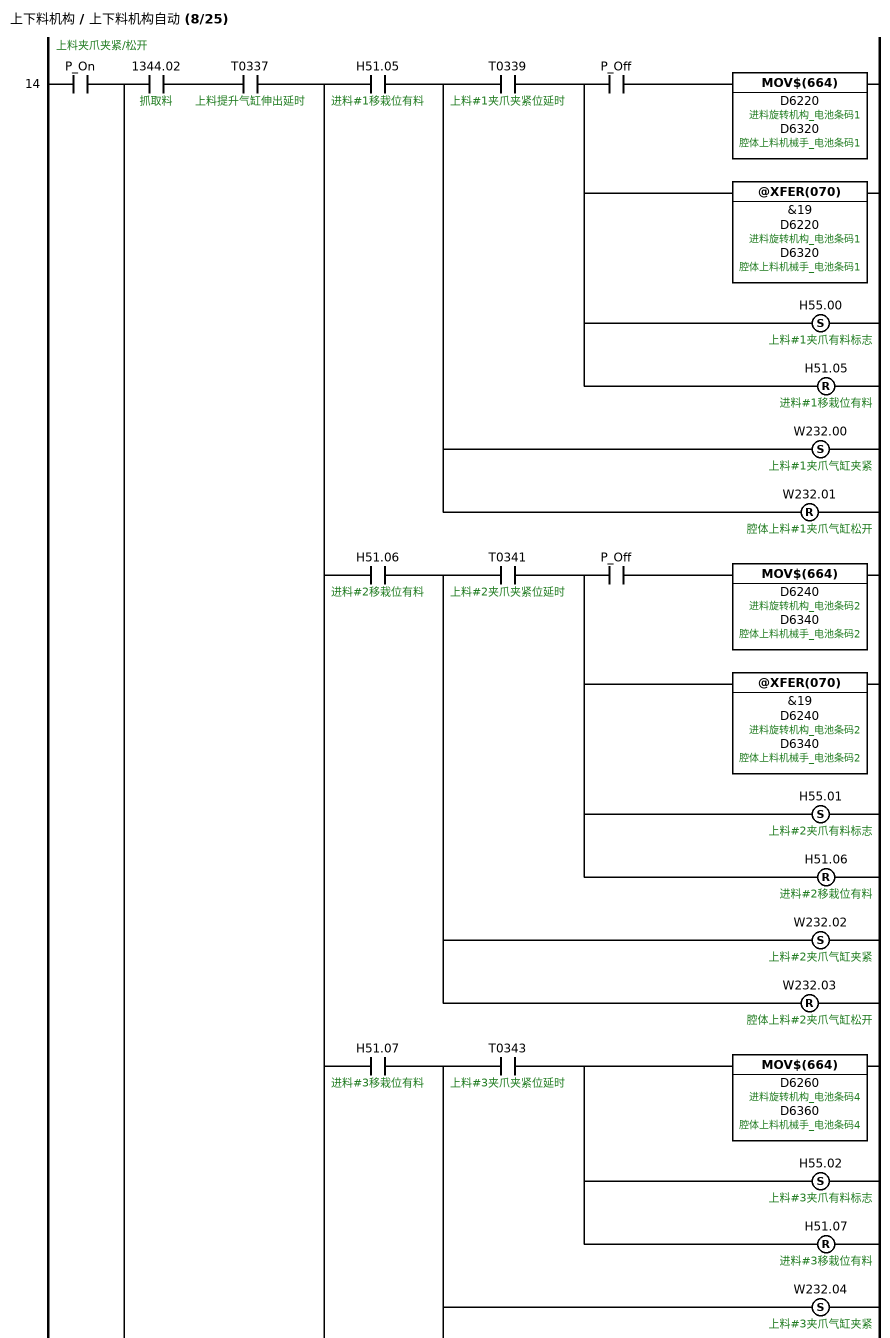
; [picture p168: 上下料机构 / 上下料机构自动, rungs 14-14]

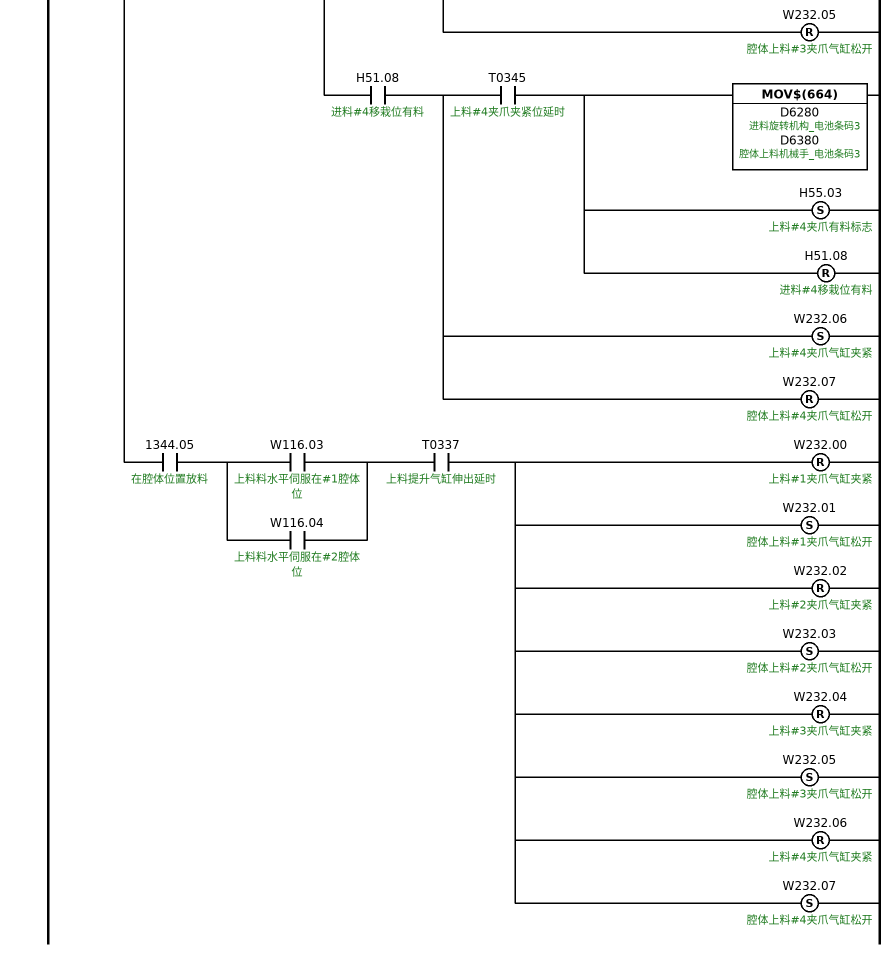
; rung 14: 上料夹爪夹紧/松开
LD P_On
OUT TR0
AND 1344.02  ; 抓取料
AND T0337  ; 上料提升气缸伸出延时
OUT TR1
AND H51.05  ; 进料#1移栽位有料
OUT TR2
AND T0339  ; 上料#1夹爪夹紧位延时
OUT TR3
AND P_Off
MOV$(664) D6220 D6320  ; 进料旋转机构_电池条码1, 腔体上料机械手_电池条码1
LD TR3
@XFER(070) &19 D6220 D6320  ; 进料旋转机构_电池条码1, 腔体上料机械手_电池条码1
SET H55.00  ; 上料#1夹爪有料标志
RSET H51.05  ; 进料#1移栽位有料
LD TR2
SET W232.00  ; 上料#1夹爪气缸夹紧
RSET W232.01  ; 腔体上料#1夹爪气缸松开
LD TR1
AND H51.06  ; 进料#2移栽位有料
OUT TR2
AND T0341  ; 上料#2夹爪夹紧位延时
OUT TR3
AND P_Off
MOV$(664) D6240 D6340  ; 进料旋转机构_电池条码2, 腔体上料机械手_电池条码2
LD TR3
@XFER(070) &19 D6240 D6340  ; 进料旋转机构_电池条码2, 腔体上料机械手_电池条码2
SET H55.01  ; 上料#2夹爪有料标志
RSET H51.06  ; 进料#2移栽位有料
LD TR2
SET W232.02  ; 上料#2夹爪气缸夹紧
RSET W232.03  ; 腔体上料#2夹爪气缸松开
LD TR1
AND H51.07  ; 进料#3移栽位有料
OUT TR2
AND T0343  ; 上料#3夹爪夹紧位延时
MOV$(664) D6260 D6360  ; 进料旋转机构_电池条码4, 腔体上料机械手_电池条码4
SET H55.02  ; 上料#3夹爪有料标志
RSET H51.07  ; 进料#3移栽位有料
LD TR2
SET W232.04  ; 上料#3夹爪气缸夹紧
RSET W232.05  ; 腔体上料#3夹爪气缸松开
LD TR1
AND H51.08  ; 进料#4移栽位有料
OUT TR1
AND T0345  ; 上料#4夹爪夹紧位延时
MOV$(664) D6280 D6380  ; 进料旋转机构_电池条码3, 腔体上料机械手_电池条码3
SET H55.03  ; 上料#4夹爪有料标志
RSET H51.08  ; 进料#4移栽位有料
LD TR1
SET W232.06  ; 上料#4夹爪气缸夹紧
RSET W232.07  ; 腔体上料#4夹爪气缸松开
LD TR0
AND 1344.05  ; 在腔体位置放料
LD W116.03  ; 上料料水平伺服在#1腔体位
OR W116.04  ; 上料料水平伺服在#2腔体位
ANDLD
AND T0337  ; 上料提升气缸伸出延时
RSET W232.00  ; 上料#1夹爪气缸夹紧
SET W232.01  ; 腔体上料#1夹爪气缸松开
RSET W232.02  ; 上料#2夹爪气缸夹紧
SET W232.03  ; 腔体上料#2夹爪气缸松开
RSET W232.04  ; 上料#3夹爪气缸夹紧
SET W232.05  ; 腔体上料#3夹爪气缸松开
RSET W232.06  ; 上料#4夹爪气缸夹紧
SET W232.07  ; 腔体上料#4夹爪气缸松开

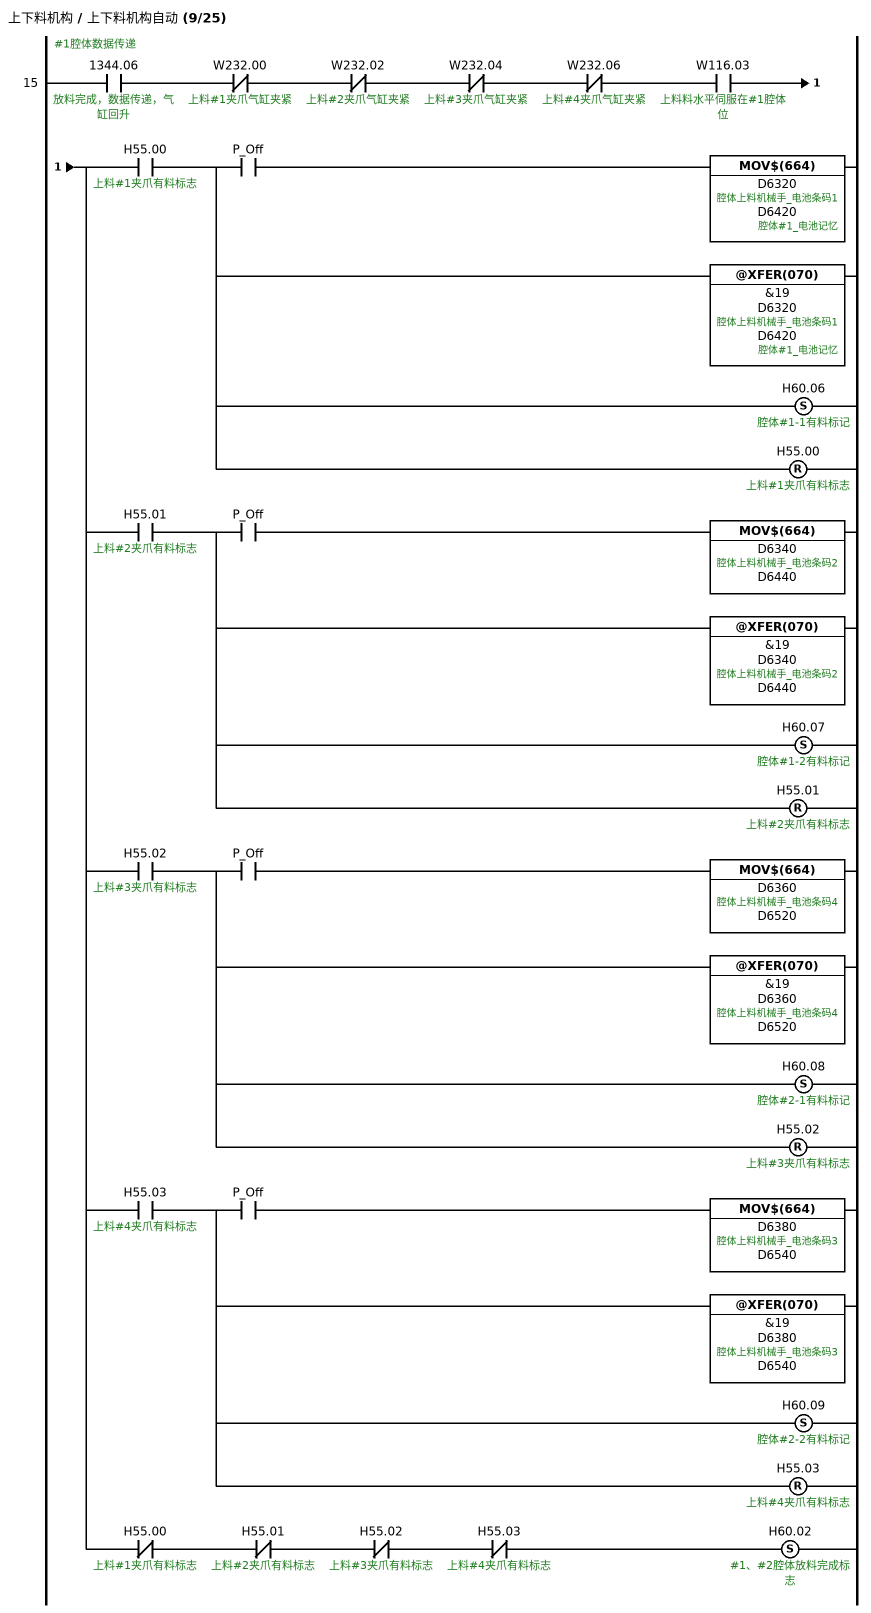
; rung 15: #1腔体数据传递
LD 1344.06  ; 放料完成，数据传递，气缸回升
ANDNOT W232.00  ; 上料#1夹爪气缸夹紧
ANDNOT W232.02  ; 上料#2夹爪气缸夹紧
ANDNOT W232.04  ; 上料#3夹爪气缸夹紧
ANDNOT W232.06  ; 上料#4夹爪气缸夹紧
AND W116.03  ; 上料料水平伺服在#1腔体位
OUT TR0
AND H55.00  ; 上料#1夹爪有料标志
OUT TR1
AND P_Off
MOV$(664) D6320 D6420  ; 腔体上料机械手_电池条码1, 腔体#1_电池记忆
LD TR1
@XFER(070) &19 D6320 D6420  ; 腔体上料机械手_电池条码1, 腔体#1_电池记忆
SET H60.06  ; 腔体#1-1有料标记
RSET H55.00  ; 上料#1夹爪有料标志
LD TR0
AND H55.01  ; 上料#2夹爪有料标志
OUT TR1
AND P_Off
MOV$(664) D6340 D6440  ; 腔体上料机械手_电池条码2
LD TR1
@XFER(070) &19 D6340 D6440  ; 腔体上料机械手_电池条码2
SET H60.07  ; 腔体#1-2有料标记
RSET H55.01  ; 上料#2夹爪有料标志
LD TR0
AND H55.02  ; 上料#3夹爪有料标志
OUT TR1
AND P_Off
MOV$(664) D6360 D6520  ; 腔体上料机械手_电池条码4
LD TR1
@XFER(070) &19 D6360 D6520  ; 腔体上料机械手_电池条码4
SET H60.08  ; 腔体#2-1有料标记
RSET H55.02  ; 上料#3夹爪有料标志
LD TR0
AND H55.03  ; 上料#4夹爪有料标志
OUT TR1
AND P_Off
MOV$(664) D6380 D6540  ; 腔体上料机械手_电池条码3
LD TR1
@XFER(070) &19 D6380 D6540  ; 腔体上料机械手_电池条码3
SET H60.09  ; 腔体#2-2有料标记
RSET H55.03  ; 上料#4夹爪有料标志
LD TR0
ANDNOT H55.00  ; 上料#1夹爪有料标志
ANDNOT H55.01  ; 上料#2夹爪有料标志
ANDNOT H55.02  ; 上料#3夹爪有料标志
ANDNOT H55.03  ; 上料#4夹爪有料标志
SET H60.02  ; #1、#2腔体放料完成标志

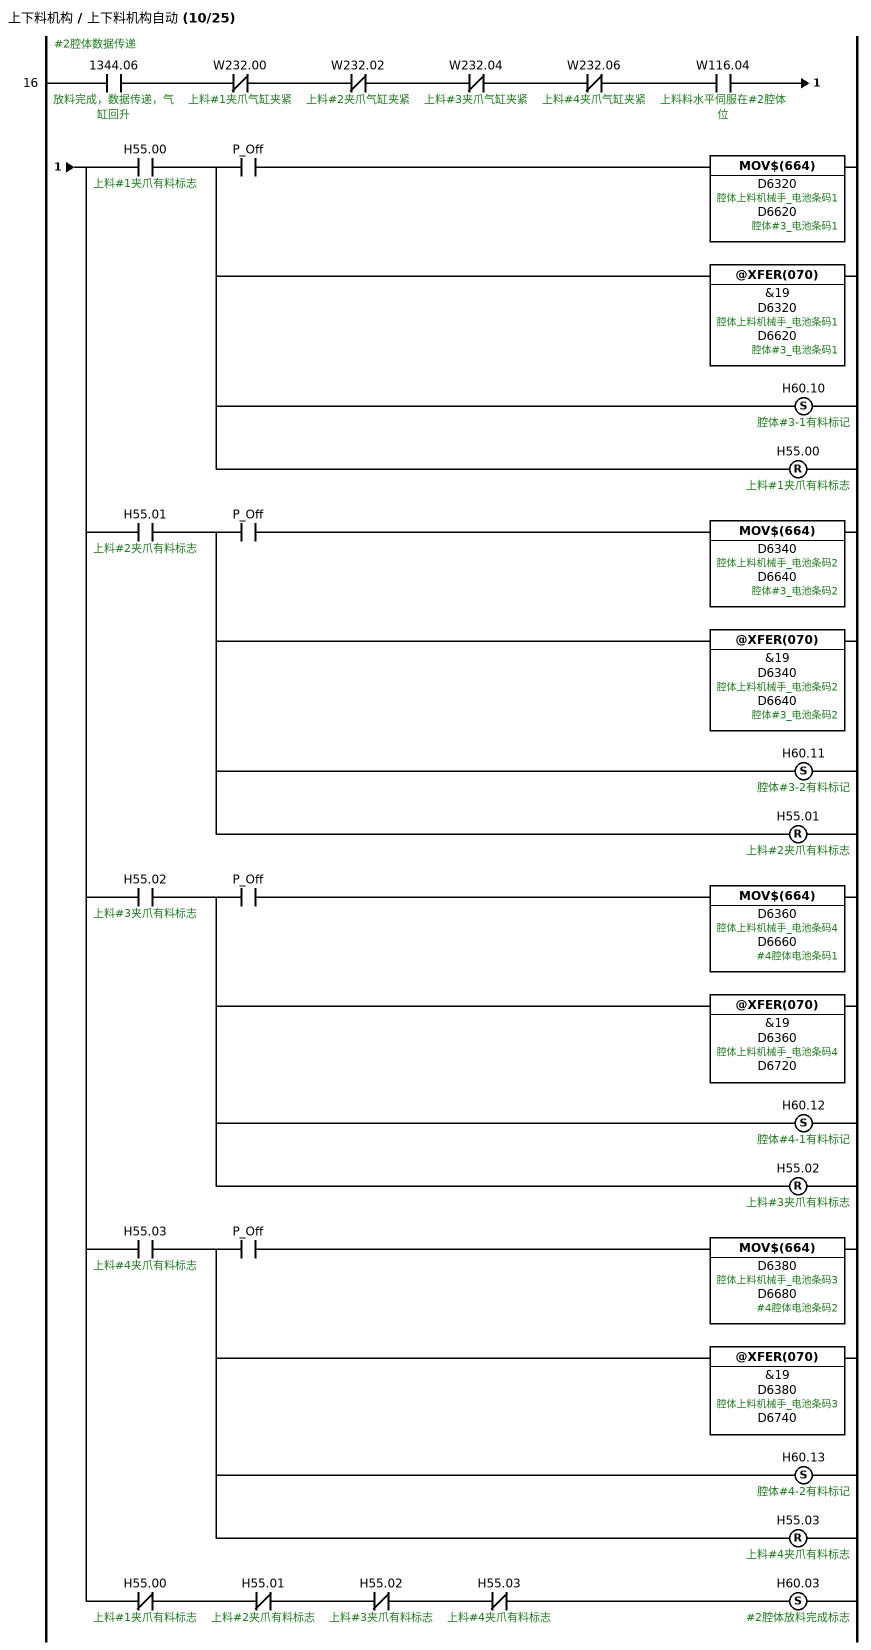
; rung 16: #2腔体数据传递
LD 1344.06  ; 放料完成，数据传递，气缸回升
ANDNOT W232.00  ; 上料#1夹爪气缸夹紧
ANDNOT W232.02  ; 上料#2夹爪气缸夹紧
ANDNOT W232.04  ; 上料#3夹爪气缸夹紧
ANDNOT W232.06  ; 上料#4夹爪气缸夹紧
AND W116.04  ; 上料料水平伺服在#2腔体位
OUT TR0
AND H55.00  ; 上料#1夹爪有料标志
OUT TR1
AND P_Off
MOV$(664) D6320 D6620  ; 腔体上料机械手_电池条码1, 腔体#3_电池条码1
LD TR1
@XFER(070) &19 D6320 D6620  ; 腔体上料机械手_电池条码1, 腔体#3_电池条码1
SET H60.10  ; 腔体#3-1有料标记
RSET H55.00  ; 上料#1夹爪有料标志
LD TR0
AND H55.01  ; 上料#2夹爪有料标志
OUT TR1
AND P_Off
MOV$(664) D6340 D6640  ; 腔体上料机械手_电池条码2, 腔体#3_电池条码2
LD TR1
@XFER(070) &19 D6340 D6640  ; 腔体上料机械手_电池条码2, 腔体#3_电池条码2
SET H60.11  ; 腔体#3-2有料标记
RSET H55.01  ; 上料#2夹爪有料标志
LD TR0
AND H55.02  ; 上料#3夹爪有料标志
OUT TR1
AND P_Off
MOV$(664) D6360 D6660  ; 腔体上料机械手_电池条码4, #4腔体电池条码1
LD TR1
@XFER(070) &19 D6360 D6720  ; 腔体上料机械手_电池条码4
SET H60.12  ; 腔体#4-1有料标记
RSET H55.02  ; 上料#3夹爪有料标志
LD TR0
AND H55.03  ; 上料#4夹爪有料标志
OUT TR1
AND P_Off
MOV$(664) D6380 D6680  ; 腔体上料机械手_电池条码3, #4腔体电池条码2
LD TR1
@XFER(070) &19 D6380 D6740  ; 腔体上料机械手_电池条码3
SET H60.13  ; 腔体#4-2有料标记
RSET H55.03  ; 上料#4夹爪有料标志
LD TR0
ANDNOT H55.00  ; 上料#1夹爪有料标志
ANDNOT H55.01  ; 上料#2夹爪有料标志
ANDNOT H55.02  ; 上料#3夹爪有料标志
ANDNOT H55.03  ; 上料#4夹爪有料标志
SET H60.03  ; #2腔体放料完成标志

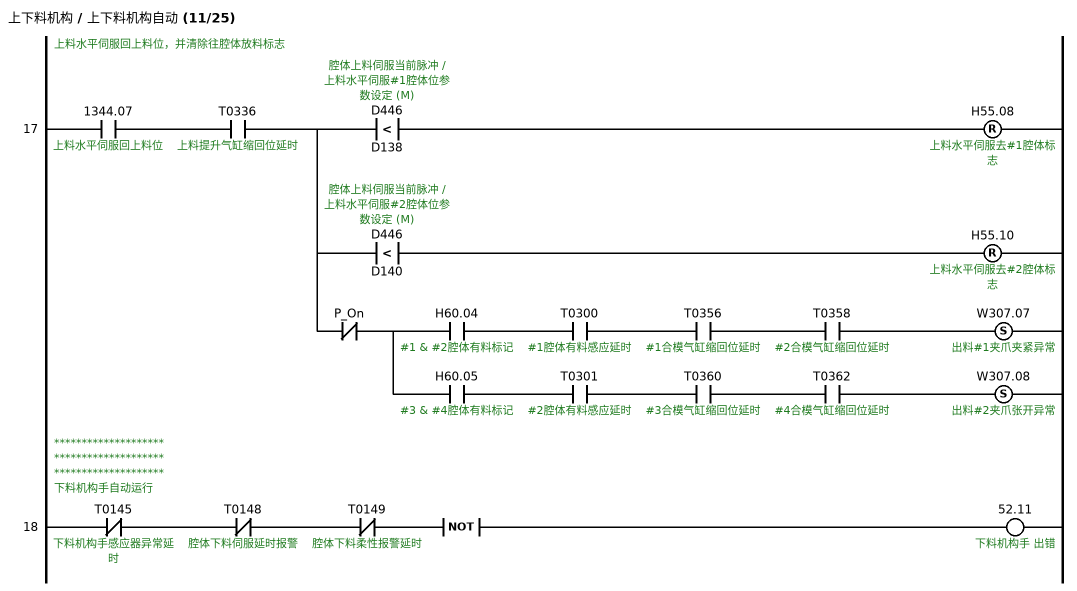
; rung 17: 上料水平伺服回上料位，并清除往腔体放料标志
LD 1344.07  ; 上料水平伺服回上料位
AND T0336  ; 上料提升气缸缩回位延时
OUT TR0
AND<F(331) D446 D138  ; 腔体上料伺服当前脉冲, 上料水平伺服#1腔体位参数设定 (M)
RSET H55.08  ; 上料水平伺服去#1腔体标志
LD TR0
AND<F(331) D446 D140  ; 腔体上料伺服当前脉冲, 上料水平伺服#2腔体位参数设定 (M)
RSET H55.10  ; 上料水平伺服去#2腔体标志
LD TR0
ANDNOT P_On
OUT TR0
AND H60.04  ; #1 & #2腔体有料标记
AND T0300  ; #1腔体有料感应延时
AND T0356  ; #1合模气缸缩回位延时
AND T0358  ; #2合模气缸缩回位延时
SET W307.07  ; 出料#1夹爪夹紧异常
LD TR0
AND H60.05  ; #3 & #4腔体有料标记
AND T0301  ; #2腔体有料感应延时
AND T0360  ; #3合模气缸缩回位延时
AND T0362  ; #4合模气缸缩回位延时
SET W307.08  ; 出料#2夹爪张开异常
; rung 18: ******************** / ******************** / ******************** / 下料机构手自动运行
LDNOT T0145  ; 下料机构手感应器异常延时
ANDNOT T0148  ; 腔体下料伺服延时报警
ANDNOT T0149  ; 腔体下料柔性报警延时
NOT(520)
OUT 52.11  ; 下料机构手 出错

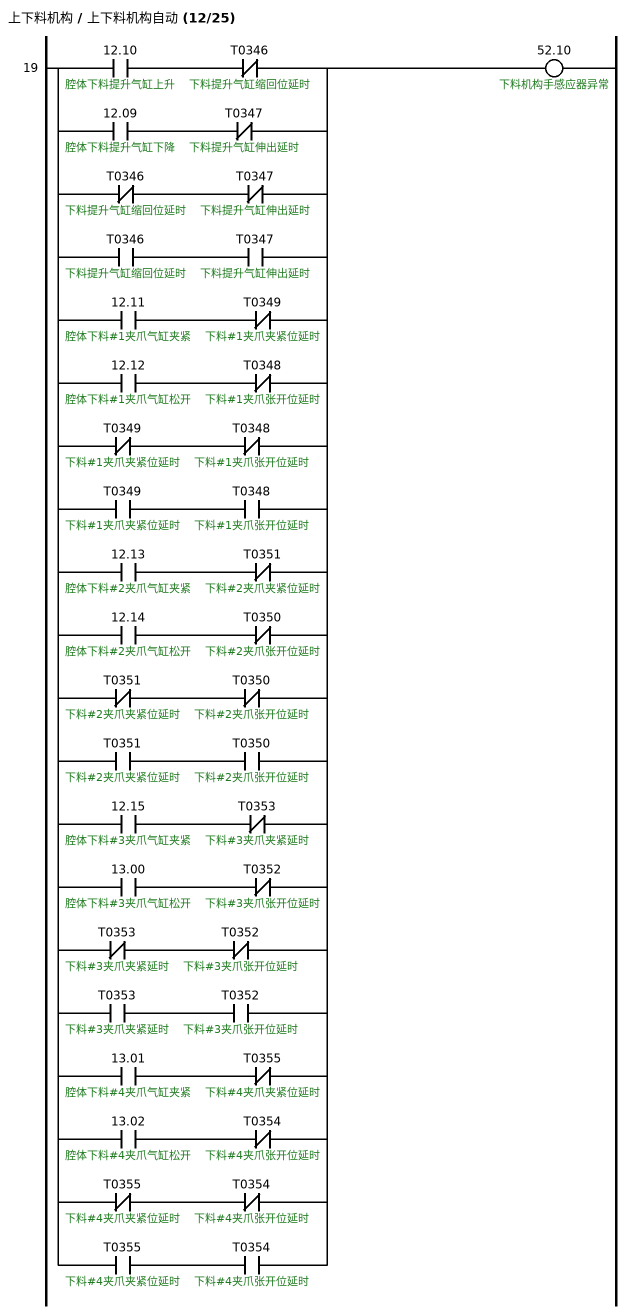
; rung 19
LD 12.10  ; 腔体下料提升气缸上升
ANDNOT T0346  ; 下料提升气缸缩回位延时
LD 12.09  ; 腔体下料提升气缸下降
ANDNOT T0347  ; 下料提升气缸伸出延时
ORLD
LDNOT T0346  ; 下料提升气缸缩回位延时
ANDNOT T0347  ; 下料提升气缸伸出延时
ORLD
LD T0346  ; 下料提升气缸缩回位延时
AND T0347  ; 下料提升气缸伸出延时
ORLD
LD 12.11  ; 腔体下料#1夹爪气缸夹紧
ANDNOT T0349  ; 下料#1夹爪夹紧位延时
ORLD
LD 12.12  ; 腔体下料#1夹爪气缸松开
ANDNOT T0348  ; 下料#1夹爪张开位延时
ORLD
LDNOT T0349  ; 下料#1夹爪夹紧位延时
ANDNOT T0348  ; 下料#1夹爪张开位延时
ORLD
LD T0349  ; 下料#1夹爪夹紧位延时
AND T0348  ; 下料#1夹爪张开位延时
ORLD
LD 12.13  ; 腔体下料#2夹爪气缸夹紧
ANDNOT T0351  ; 下料#2夹爪夹紧位延时
ORLD
LD 12.14  ; 腔体下料#2夹爪气缸松开
ANDNOT T0350  ; 下料#2夹爪张开位延时
ORLD
LDNOT T0351  ; 下料#2夹爪夹紧位延时
ANDNOT T0350  ; 下料#2夹爪张开位延时
ORLD
LD T0351  ; 下料#2夹爪夹紧位延时
AND T0350  ; 下料#2夹爪张开位延时
ORLD
LD 12.15  ; 腔体下料#3夹爪气缸夹紧
ANDNOT T0353  ; 下料#3夹爪夹紧延时
ORLD
LD 13.00  ; 腔体下料#3夹爪气缸松开
ANDNOT T0352  ; 下料#3夹爪张开位延时
ORLD
LDNOT T0353  ; 下料#3夹爪夹紧延时
ANDNOT T0352  ; 下料#3夹爪张开位延时
ORLD
LD T0353  ; 下料#3夹爪夹紧延时
AND T0352  ; 下料#3夹爪张开位延时
ORLD
LD 13.01  ; 腔体下料#4夹爪气缸夹紧
ANDNOT T0355  ; 下料#4夹爪夹紧位延时
ORLD
LD 13.02  ; 腔体下料#4夹爪气缸松开
ANDNOT T0354  ; 下料#4夹爪张开位延时
ORLD
LDNOT T0355  ; 下料#4夹爪夹紧位延时
ANDNOT T0354  ; 下料#4夹爪张开位延时
ORLD
LD T0355  ; 下料#4夹爪夹紧位延时
AND T0354  ; 下料#4夹爪张开位延时
ORLD
OUT 52.10  ; 下料机构手感应器异常

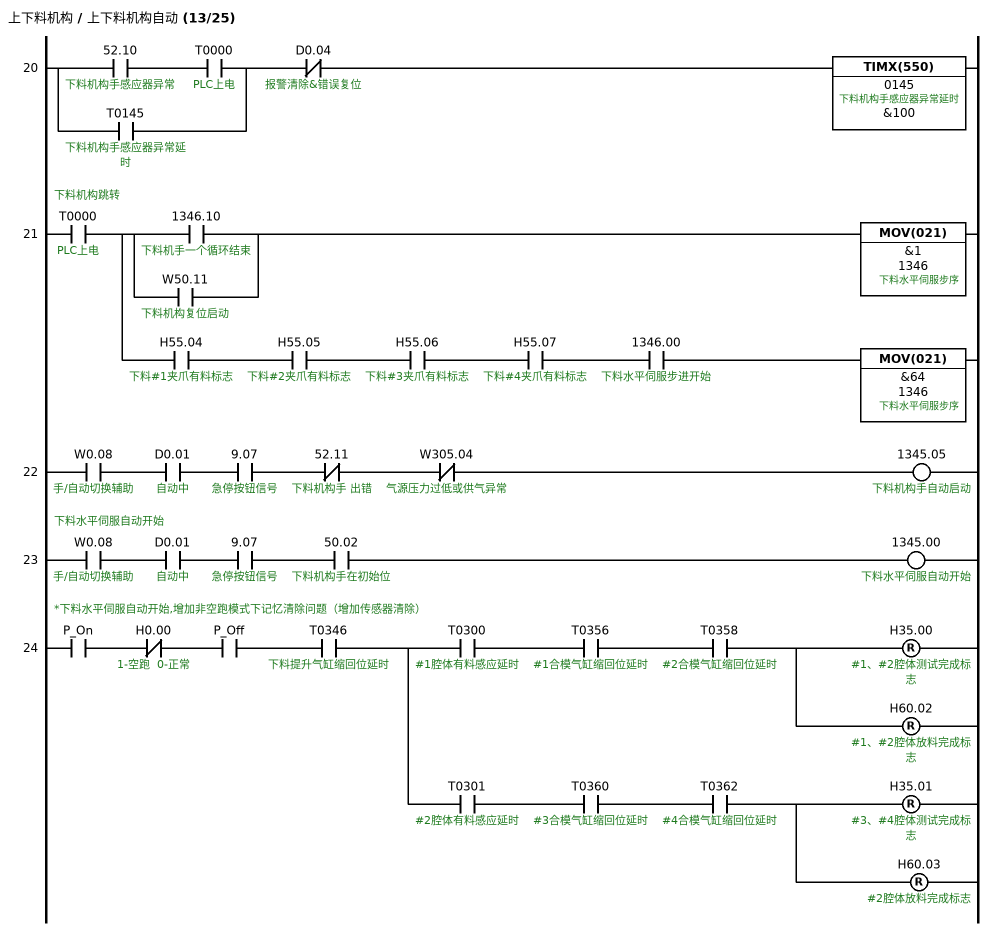
; rung 20
LD 52.10  ; 下料机构手感应器异常
AND T0000  ; PLC上电
OR T0145  ; 下料机构手感应器异常延时
ANDNOT D0.04  ; 报警清除&错误复位
TIMX(550) 0145 &100  ; 下料机构手感应器异常延时
; rung 21: 下料机构跳转
LD T0000  ; PLC上电
OUT TR0
LD 1346.10  ; 下料机手一个循环结束
OR W50.11  ; 下料机构复位启动
ANDLD
MOV(021) &1 1346  ; 下料水平伺服步序
LD TR0
AND H55.04  ; 下料#1夹爪有料标志
AND H55.05  ; 下料#2夹爪有料标志
AND H55.06  ; 下料#3夹爪有料标志
AND H55.07  ; 下料#4夹爪有料标志
AND 1346.00  ; 下料水平伺服步进开始
MOV(021) &64 1346  ; 下料水平伺服步序
; rung 22
LD W0.08  ; 手/自动切换辅助
AND D0.01  ; 自动中
AND 9.07  ; 急停按钮信号
ANDNOT 52.11  ; 下料机构手 出错
ANDNOT W305.04  ; 气源压力过低或供气异常
OUT 1345.05  ; 下料机构手自动启动
; rung 23: 下料水平伺服自动开始
LD W0.08  ; 手/自动切换辅助
AND D0.01  ; 自动中
AND 9.07  ; 急停按钮信号
AND 50.02  ; 下料机构手在初始位
OUT 1345.00  ; 下料水平伺服自动开始
; rung 24: *下料水平伺服自动开始,增加非空跑模式下记忆清除问题（增加传感器清除）
LD P_On
ANDNOT H0.00  ; 1-空跑  0-正常
AND P_Off
AND T0346  ; 下料提升气缸缩回位延时
OUT TR0
AND T0300  ; #1腔体有料感应延时
AND T0356  ; #1合模气缸缩回位延时
AND T0358  ; #2合模气缸缩回位延时
RSET H35.00  ; #1、#2腔体测试完成标志
RSET H60.02  ; #1、#2腔体放料完成标志
LD TR0
AND T0301  ; #2腔体有料感应延时
AND T0360  ; #3合模气缸缩回位延时
AND T0362  ; #4合模气缸缩回位延时
RSET H35.01  ; #3、#4腔体测试完成标志
RSET H60.03  ; #2腔体放料完成标志

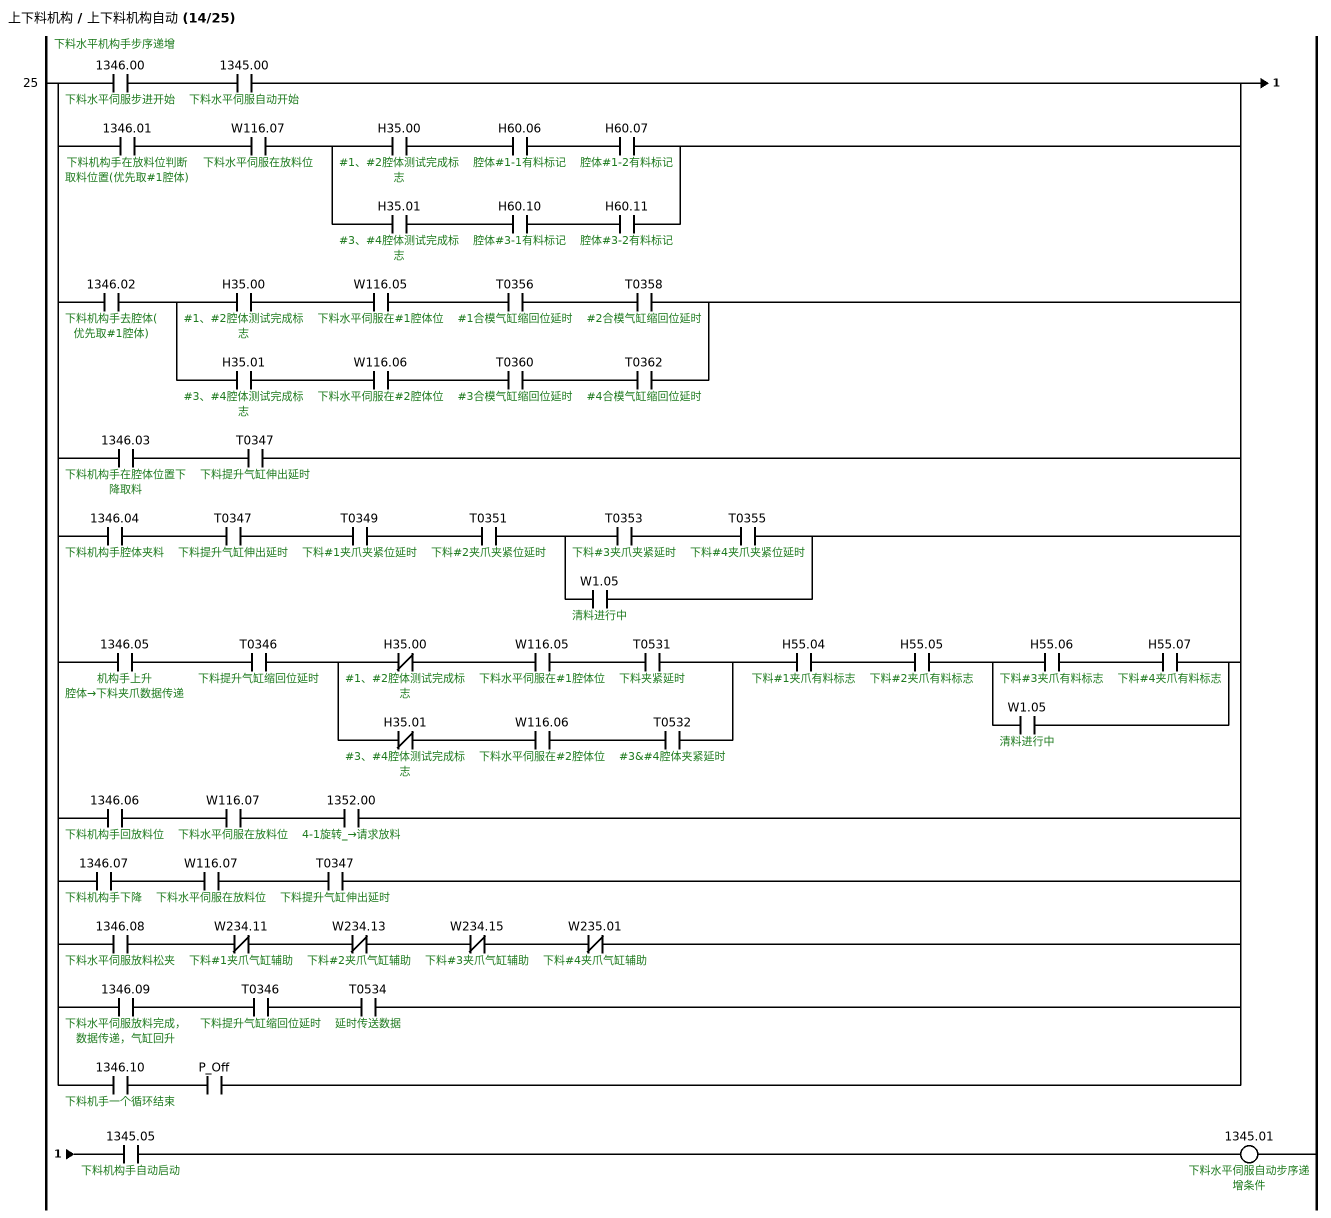
; rung 25: 下料水平机构手步序递增
LD 1346.00  ; 下料水平伺服步进开始
AND 1345.00  ; 下料水平伺服自动开始
LD 1346.01  ; 下料机构手在放料位判断取料位置(优先取#1腔体)
AND W116.07  ; 下料水平伺服在放料位
LD H35.00  ; #1、#2腔体测试完成标志
AND H60.06  ; 腔体#1-1有料标记
AND H60.07  ; 腔体#1-2有料标记
LD H35.01  ; #3、#4腔体测试完成标志
AND H60.10  ; 腔体#3-1有料标记
AND H60.11  ; 腔体#3-2有料标记
ORLD
ANDLD
ORLD
LD 1346.02  ; 下料机构手去腔体(优先取#1腔体)
LD H35.00  ; #1、#2腔体测试完成标志
AND W116.05  ; 下料水平伺服在#1腔体位
AND T0356  ; #1合模气缸缩回位延时
AND T0358  ; #2合模气缸缩回位延时
LD H35.01  ; #3、#4腔体测试完成标志
AND W116.06  ; 下料水平伺服在#2腔体位
AND T0360  ; #3合模气缸缩回位延时
AND T0362  ; #4合模气缸缩回位延时
ORLD
ANDLD
ORLD
LD 1346.03  ; 下料机构手在腔体位置下降取料
AND T0347  ; 下料提升气缸伸出延时
ORLD
LD 1346.04  ; 下料机构手腔体夹料
AND T0347  ; 下料提升气缸伸出延时
AND T0349  ; 下料#1夹爪夹紧位延时
AND T0351  ; 下料#2夹爪夹紧位延时
LD T0353  ; 下料#3夹爪夹紧延时
AND T0355  ; 下料#4夹爪夹紧位延时
OR W1.05  ; 清料进行中
ANDLD
ORLD
LD 1346.05  ; 机构手上升 腔体→下料夹爪数据传递
AND T0346  ; 下料提升气缸缩回位延时
LDNOT H35.00  ; #1、#2腔体测试完成标志
AND W116.05  ; 下料水平伺服在#1腔体位
AND T0531  ; 下料夹紧延时
LDNOT H35.01  ; #3、#4腔体测试完成标志
AND W116.06  ; 下料水平伺服在#2腔体位
AND T0532  ; #3&#4腔体夹紧延时
ORLD
ANDLD
AND H55.04  ; 下料#1夹爪有料标志
AND H55.05  ; 下料#2夹爪有料标志
LD H55.06  ; 下料#3夹爪有料标志
AND H55.07  ; 下料#4夹爪有料标志
OR W1.05  ; 清料进行中
ANDLD
ORLD
LD 1346.06  ; 下料机构手回放料位
AND W116.07  ; 下料水平伺服在放料位
AND 1352.00  ; 4-1旋转_→请求放料
ORLD
LD 1346.07  ; 下料机构手下降
AND W116.07  ; 下料水平伺服在放料位
AND T0347  ; 下料提升气缸伸出延时
ORLD
LD 1346.08  ; 下料水平伺服放料松夹
ANDNOT W234.11  ; 下料#1夹爪气缸辅助
ANDNOT W234.13  ; 下料#2夹爪气缸辅助
ANDNOT W234.15  ; 下料#3夹爪气缸辅助
ANDNOT W235.01  ; 下料#4夹爪气缸辅助
ORLD
LD 1346.09  ; 下料水平伺服放料完成，数据传递，气缸回升
AND T0346  ; 下料提升气缸缩回位延时
AND T0534  ; 延时传送数据
ORLD
LD 1346.10  ; 下料机手一个循环结束
AND P_Off
ORLD
AND 1345.05  ; 下料机构手自动启动
OUT 1345.01  ; 下料水平伺服自动步序递增条件

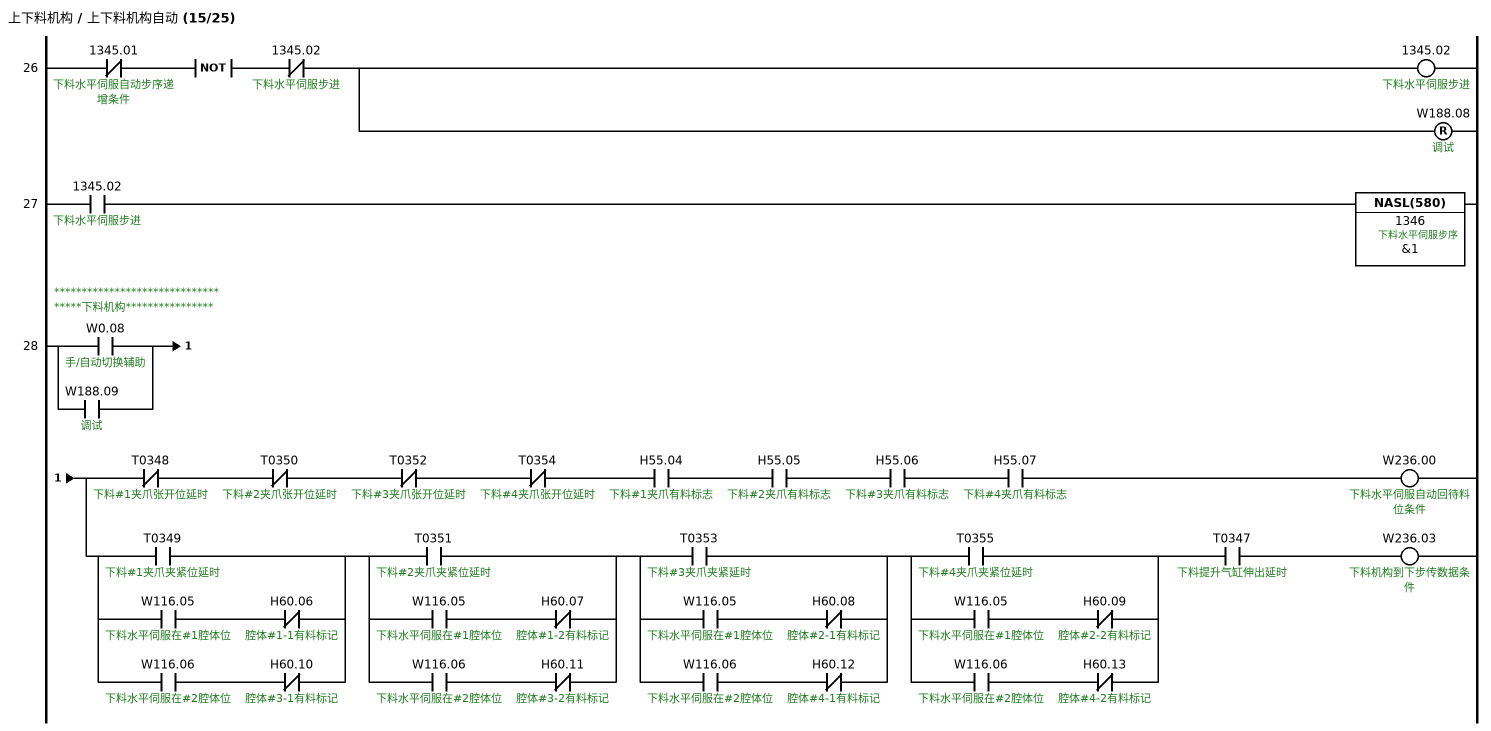
; rung 26
LDNOT 1345.01  ; 下料水平伺服自动步序递增条件
NOT(520)
ANDNOT 1345.02  ; 下料水平伺服步进
OUT 1345.02  ; 下料水平伺服步进
RSET W188.08  ; 调试
; rung 27
LD 1345.02  ; 下料水平伺服步进
NASL(580) 1346 &1  ; 下料水平伺服步序
; rung 28: ****************************** / *****下料机构****************
LD W0.08  ; 手/自动切换辅助
OR W188.09  ; 调试
OUT TR0
ANDNOT T0348  ; 下料#1夹爪张开位延时
ANDNOT T0350  ; 下料#2夹爪张开位延时
ANDNOT T0352  ; 下料#3夹爪张开位延时
ANDNOT T0354  ; 下料#4夹爪张开位延时
AND H55.04  ; 下料#1夹爪有料标志
AND H55.05  ; 下料#2夹爪有料标志
AND H55.06  ; 下料#3夹爪有料标志
AND H55.07  ; 下料#4夹爪有料标志
OUT W236.00  ; 下料水平伺服自动回待料位条件
LD TR0
LD T0349  ; 下料#1夹爪夹紧位延时
LD W116.05  ; 下料水平伺服在#1腔体位
ANDNOT H60.06  ; 腔体#1-1有料标记
ORLD
LD W116.06  ; 下料水平伺服在#2腔体位
ANDNOT H60.10  ; 腔体#3-1有料标记
ORLD
ANDLD
LD T0351  ; 下料#2夹爪夹紧位延时
LD W116.05  ; 下料水平伺服在#1腔体位
ANDNOT H60.07  ; 腔体#1-2有料标记
ORLD
LD W116.06  ; 下料水平伺服在#2腔体位
ANDNOT H60.11  ; 腔体#3-2有料标记
ORLD
ANDLD
LD T0353  ; 下料#3夹爪夹紧延时
LD W116.05  ; 下料水平伺服在#1腔体位
ANDNOT H60.08  ; 腔体#2-1有料标记
ORLD
LD W116.06  ; 下料水平伺服在#2腔体位
ANDNOT H60.12  ; 腔体#4-1有料标记
ORLD
ANDLD
LD T0355  ; 下料#4夹爪夹紧位延时
LD W116.05  ; 下料水平伺服在#1腔体位
ANDNOT H60.09  ; 腔体#2-2有料标记
ORLD
LD W116.06  ; 下料水平伺服在#2腔体位
ANDNOT H60.13  ; 腔体#4-2有料标记
ORLD
ANDLD
AND T0347  ; 下料提升气缸伸出延时
OUT W236.03  ; 下料机构到下步传数据条件

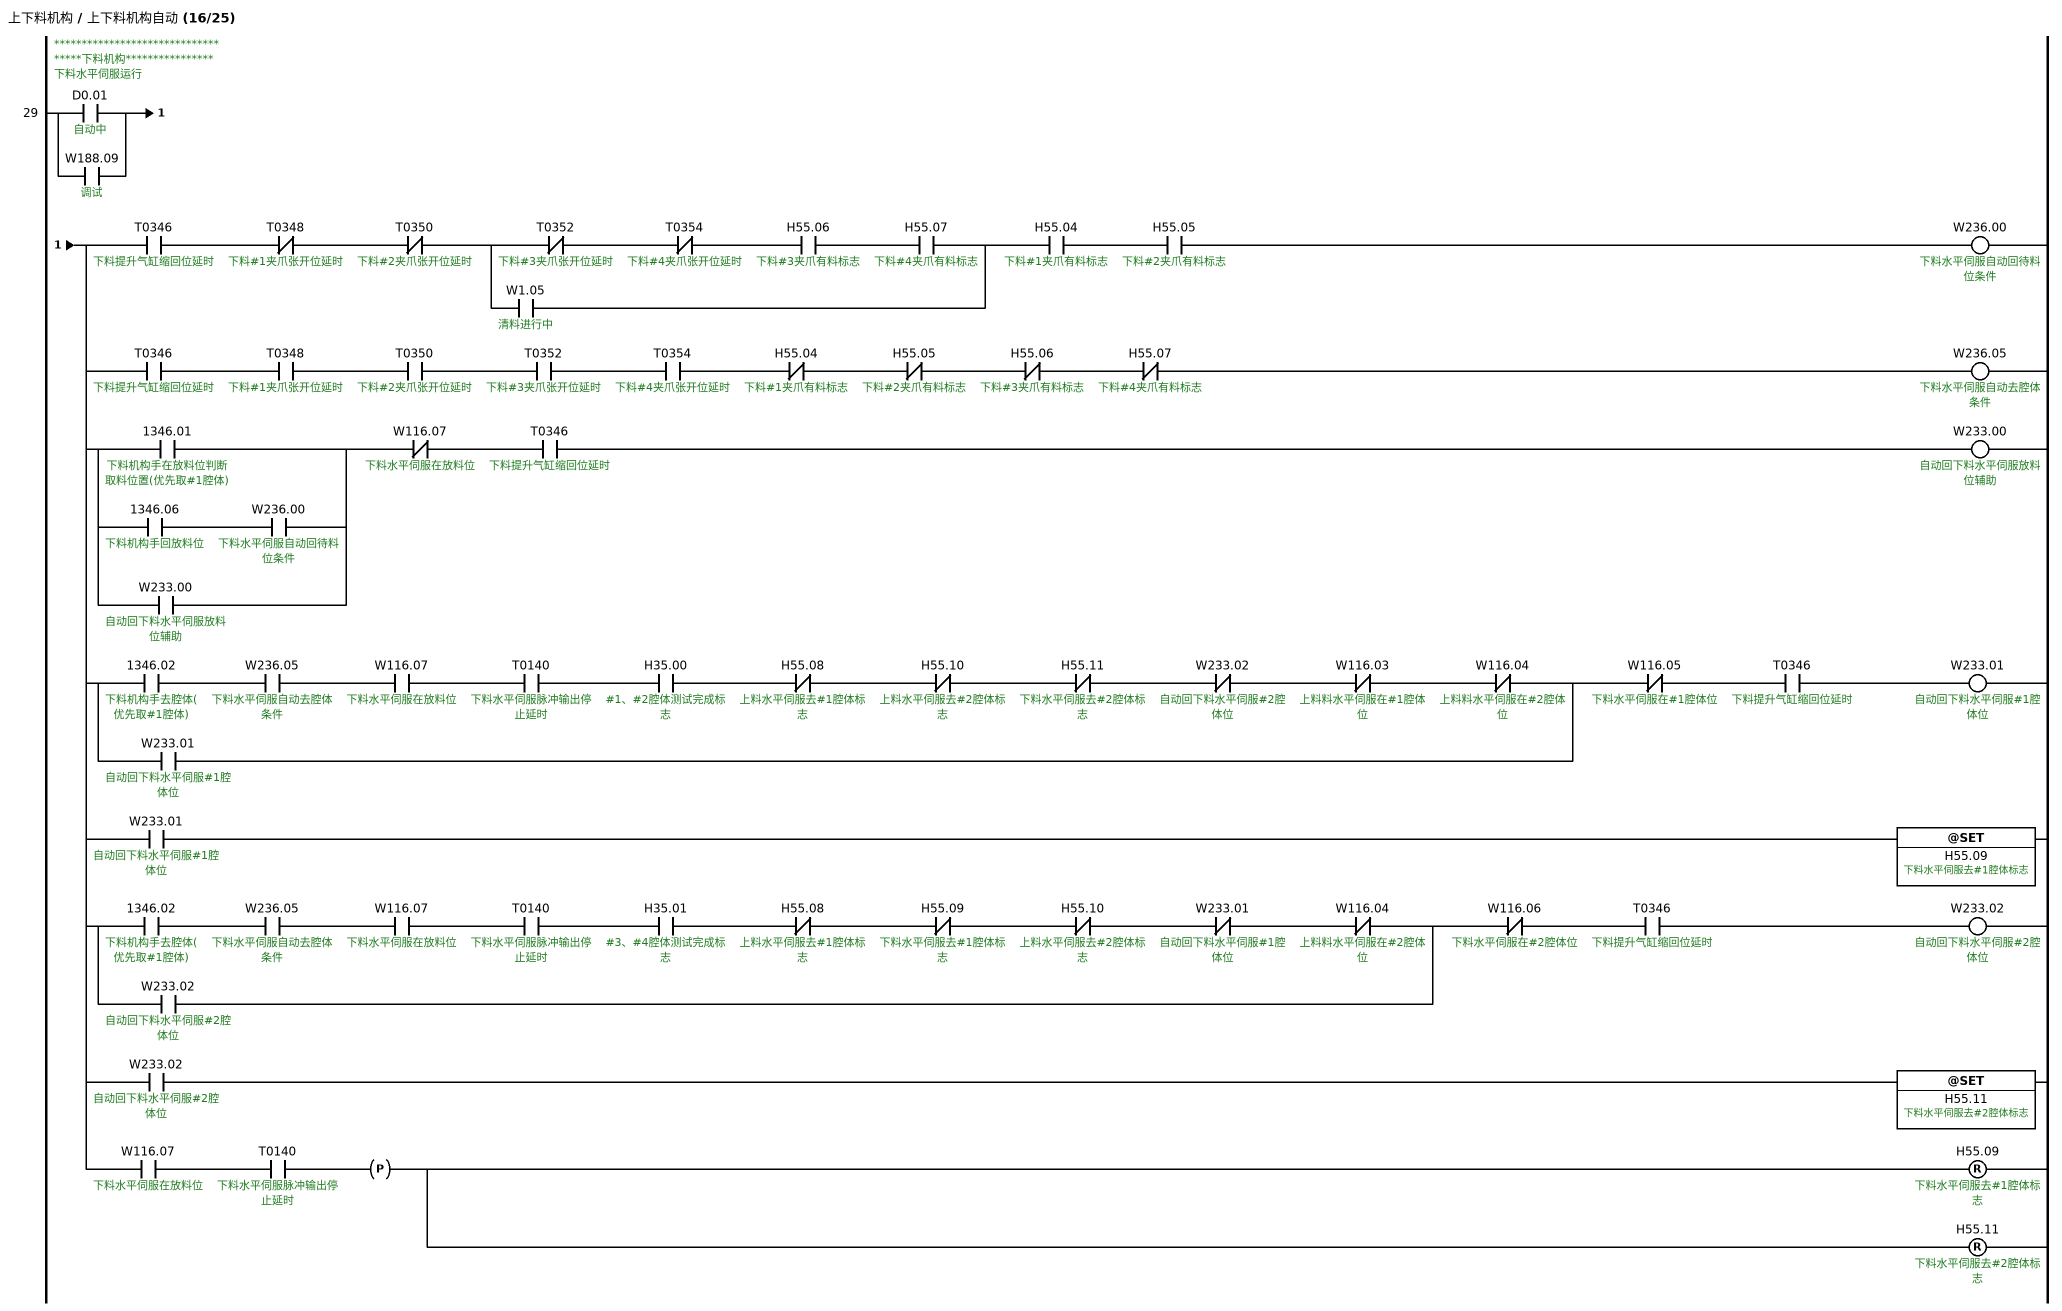
; rung 29: ****************************** / *****下料机构**************** / 下料水平伺服运行
LD D0.01  ; 自动中
OR W188.09  ; 调试
OUT TR0
AND T0346  ; 下料提升气缸缩回位延时
ANDNOT T0348  ; 下料#1夹爪张开位延时
ANDNOT T0350  ; 下料#2夹爪张开位延时
LDNOT T0352  ; 下料#3夹爪张开位延时
ANDNOT T0354  ; 下料#4夹爪张开位延时
AND H55.06  ; 下料#3夹爪有料标志
AND H55.07  ; 下料#4夹爪有料标志
OR W1.05  ; 清料进行中
ANDLD
AND H55.04  ; 下料#1夹爪有料标志
AND H55.05  ; 下料#2夹爪有料标志
OUT W236.00  ; 下料水平伺服自动回待料位条件
LD TR0
AND T0346  ; 下料提升气缸缩回位延时
AND T0348  ; 下料#1夹爪张开位延时
AND T0350  ; 下料#2夹爪张开位延时
AND T0352  ; 下料#3夹爪张开位延时
AND T0354  ; 下料#4夹爪张开位延时
ANDNOT H55.04  ; 下料#1夹爪有料标志
ANDNOT H55.05  ; 下料#2夹爪有料标志
ANDNOT H55.06  ; 下料#3夹爪有料标志
ANDNOT H55.07  ; 下料#4夹爪有料标志
OUT W236.05  ; 下料水平伺服自动去腔体条件
LD TR0
LD 1346.01  ; 下料机构手在放料位判断取料位置(优先取#1腔体)
LD 1346.06  ; 下料机构手回放料位
AND W236.00  ; 下料水平伺服自动回待料位条件
ORLD
OR W233.00  ; 自动回下料水平伺服放料位辅助
ANDLD
ANDNOT W116.07  ; 下料水平伺服在放料位
AND T0346  ; 下料提升气缸缩回位延时
OUT W233.00  ; 自动回下料水平伺服放料位辅助
LD TR0
LD 1346.02  ; 下料机构手去腔体(优先取#1腔体)
AND W236.05  ; 下料水平伺服自动去腔体条件
AND W116.07  ; 下料水平伺服在放料位
AND T0140  ; 下料水平伺服脉冲输出停止延时
AND H35.00  ; #1、#2腔体测试完成标志
ANDNOT H55.08  ; 上料水平伺服去#1腔体标志
ANDNOT H55.10  ; 上料水平伺服去#2腔体标志
ANDNOT H55.11  ; 下料水平伺服去#2腔体标志
ANDNOT W233.02  ; 自动回下料水平伺服#2腔体位
ANDNOT W116.03  ; 上料料水平伺服在#1腔体位
ANDNOT W116.04  ; 上料料水平伺服在#2腔体位
OR W233.01  ; 自动回下料水平伺服#1腔体位
ANDLD
ANDNOT W116.05  ; 下料水平伺服在#1腔体位
AND T0346  ; 下料提升气缸缩回位延时
OUT W233.01  ; 自动回下料水平伺服#1腔体位
LD TR0
AND W233.01  ; 自动回下料水平伺服#1腔体位
@SET H55.09  ; 下料水平伺服去#1腔体标志
LD TR0
LD 1346.02  ; 下料机构手去腔体(优先取#1腔体)
AND W236.05  ; 下料水平伺服自动去腔体条件
AND W116.07  ; 下料水平伺服在放料位
AND T0140  ; 下料水平伺服脉冲输出停止延时
AND H35.01  ; #3、#4腔体测试完成标志
ANDNOT H55.08  ; 上料水平伺服去#1腔体标志
ANDNOT H55.09  ; 下料水平伺服去#1腔体标志
ANDNOT H55.10  ; 上料水平伺服去#2腔体标志
ANDNOT W233.01  ; 自动回下料水平伺服#1腔体位
ANDNOT W116.04  ; 上料料水平伺服在#2腔体位
OR W233.02  ; 自动回下料水平伺服#2腔体位
ANDLD
ANDNOT W116.06  ; 下料水平伺服在#2腔体位
AND T0346  ; 下料提升气缸缩回位延时
OUT W233.02  ; 自动回下料水平伺服#2腔体位
LD TR0
AND W233.02  ; 自动回下料水平伺服#2腔体位
@SET H55.11  ; 下料水平伺服去#2腔体标志
LD TR0
AND W116.07  ; 下料水平伺服在放料位
AND T0140  ; 下料水平伺服脉冲输出停止延时
UP(521)
RSET H55.09  ; 下料水平伺服去#1腔体标志
RSET H55.11  ; 下料水平伺服去#2腔体标志

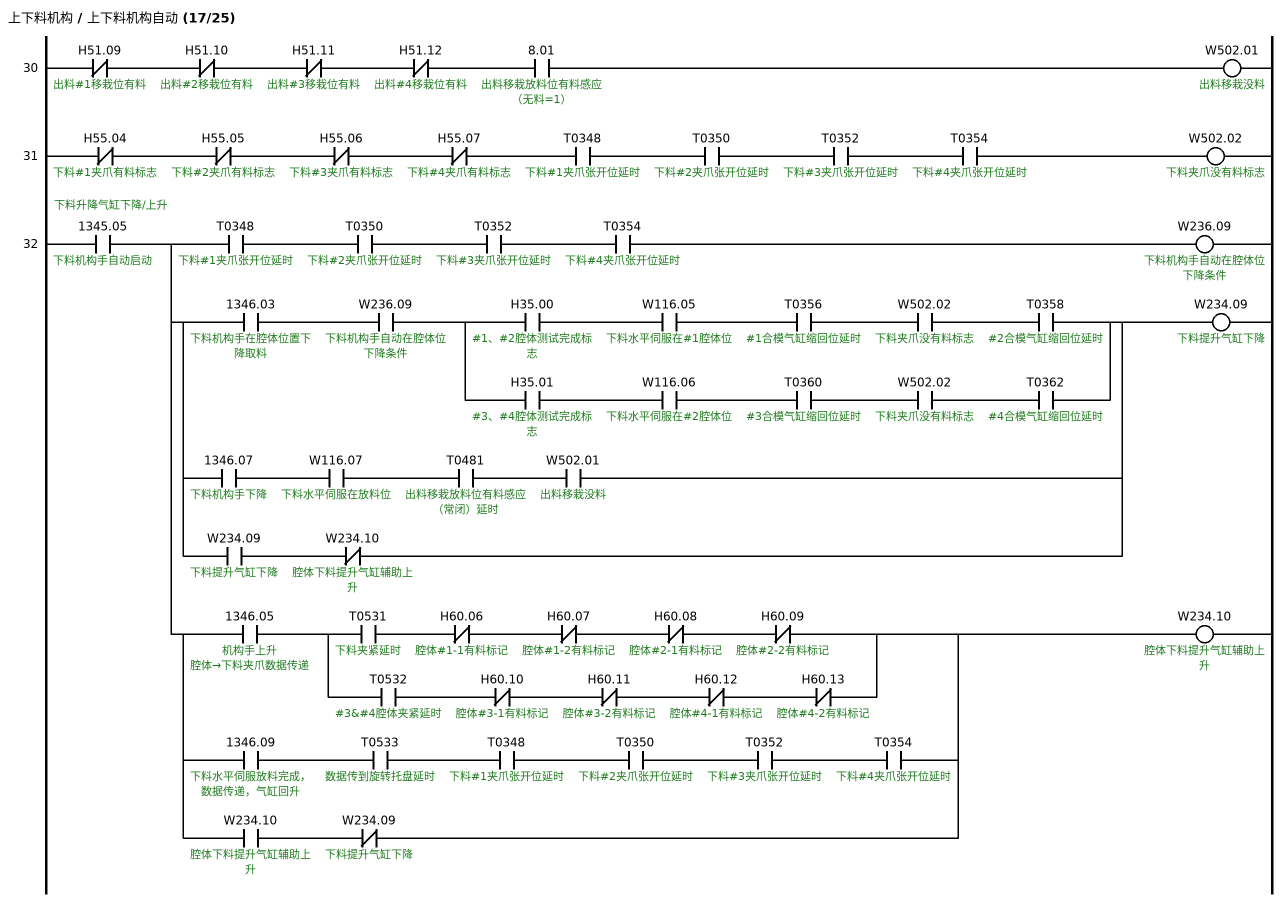
; rung 30
LDNOT H51.09  ; 出料#1移栽位有料
ANDNOT H51.10  ; 出料#2移栽位有料
ANDNOT H51.11  ; 出料#3移栽位有料
ANDNOT H51.12  ; 出料#4移栽位有料
AND 8.01  ; 出料移栽放料位有料感应（无料=1）
OUT W502.01  ; 出料移栽没料
; rung 31
LDNOT H55.04  ; 下料#1夹爪有料标志
ANDNOT H55.05  ; 下料#2夹爪有料标志
ANDNOT H55.06  ; 下料#3夹爪有料标志
ANDNOT H55.07  ; 下料#4夹爪有料标志
AND T0348  ; 下料#1夹爪张开位延时
AND T0350  ; 下料#2夹爪张开位延时
AND T0352  ; 下料#3夹爪张开位延时
AND T0354  ; 下料#4夹爪张开位延时
OUT W502.02  ; 下料夹爪没有料标志
; rung 32: 下料升降气缸下降/上升
LD 1345.05  ; 下料机构手自动启动
OUT TR0
AND T0348  ; 下料#1夹爪张开位延时
AND T0350  ; 下料#2夹爪张开位延时
AND T0352  ; 下料#3夹爪张开位延时
AND T0354  ; 下料#4夹爪张开位延时
OUT W236.09  ; 下料机构手自动在腔体位下降条件
LD TR0
LD 1346.03  ; 下料机构手在腔体位置下降取料
AND W236.09  ; 下料机构手自动在腔体位下降条件
LD H35.00  ; #1、#2腔体测试完成标志
AND W116.05  ; 下料水平伺服在#1腔体位
AND T0356  ; #1合模气缸缩回位延时
AND W502.02  ; 下料夹爪没有料标志
AND T0358  ; #2合模气缸缩回位延时
LD H35.01  ; #3、#4腔体测试完成标志
AND W116.06  ; 下料水平伺服在#2腔体位
AND T0360  ; #3合模气缸缩回位延时
AND W502.02  ; 下料夹爪没有料标志
AND T0362  ; #4合模气缸缩回位延时
ORLD
ANDLD
LD 1346.07  ; 下料机构手下降
AND W116.07  ; 下料水平伺服在放料位
AND T0481  ; 出料移栽放料位有料感应（常闭）延时
AND W502.01  ; 出料移栽没料
ORLD
LD W234.09  ; 下料提升气缸下降
ANDNOT W234.10  ; 腔体下料提升气缸辅助上升
ORLD
ANDLD
OUT W234.09  ; 下料提升气缸下降
LD TR0
LD 1346.05  ; 机构手上升 腔体→下料夹爪数据传递
LD T0531  ; 下料夹紧延时
ANDNOT H60.06  ; 腔体#1-1有料标记
ANDNOT H60.07  ; 腔体#1-2有料标记
ANDNOT H60.08  ; 腔体#2-1有料标记
ANDNOT H60.09  ; 腔体#2-2有料标记
LD T0532  ; #3&#4腔体夹紧延时
ANDNOT H60.10  ; 腔体#3-1有料标记
ANDNOT H60.11  ; 腔体#3-2有料标记
ANDNOT H60.12  ; 腔体#4-1有料标记
ANDNOT H60.13  ; 腔体#4-2有料标记
ORLD
ANDLD
LD 1346.09  ; 下料水平伺服放料完成，数据传递，气缸回升
AND T0533  ; 数据传到旋转托盘延时
AND T0348  ; 下料#1夹爪张开位延时
AND T0350  ; 下料#2夹爪张开位延时
AND T0352  ; 下料#3夹爪张开位延时
AND T0354  ; 下料#4夹爪张开位延时
ORLD
LD W234.10  ; 腔体下料提升气缸辅助上升
ANDNOT W234.09  ; 下料提升气缸下降
ORLD
ANDLD
OUT W234.10  ; 腔体下料提升气缸辅助上升

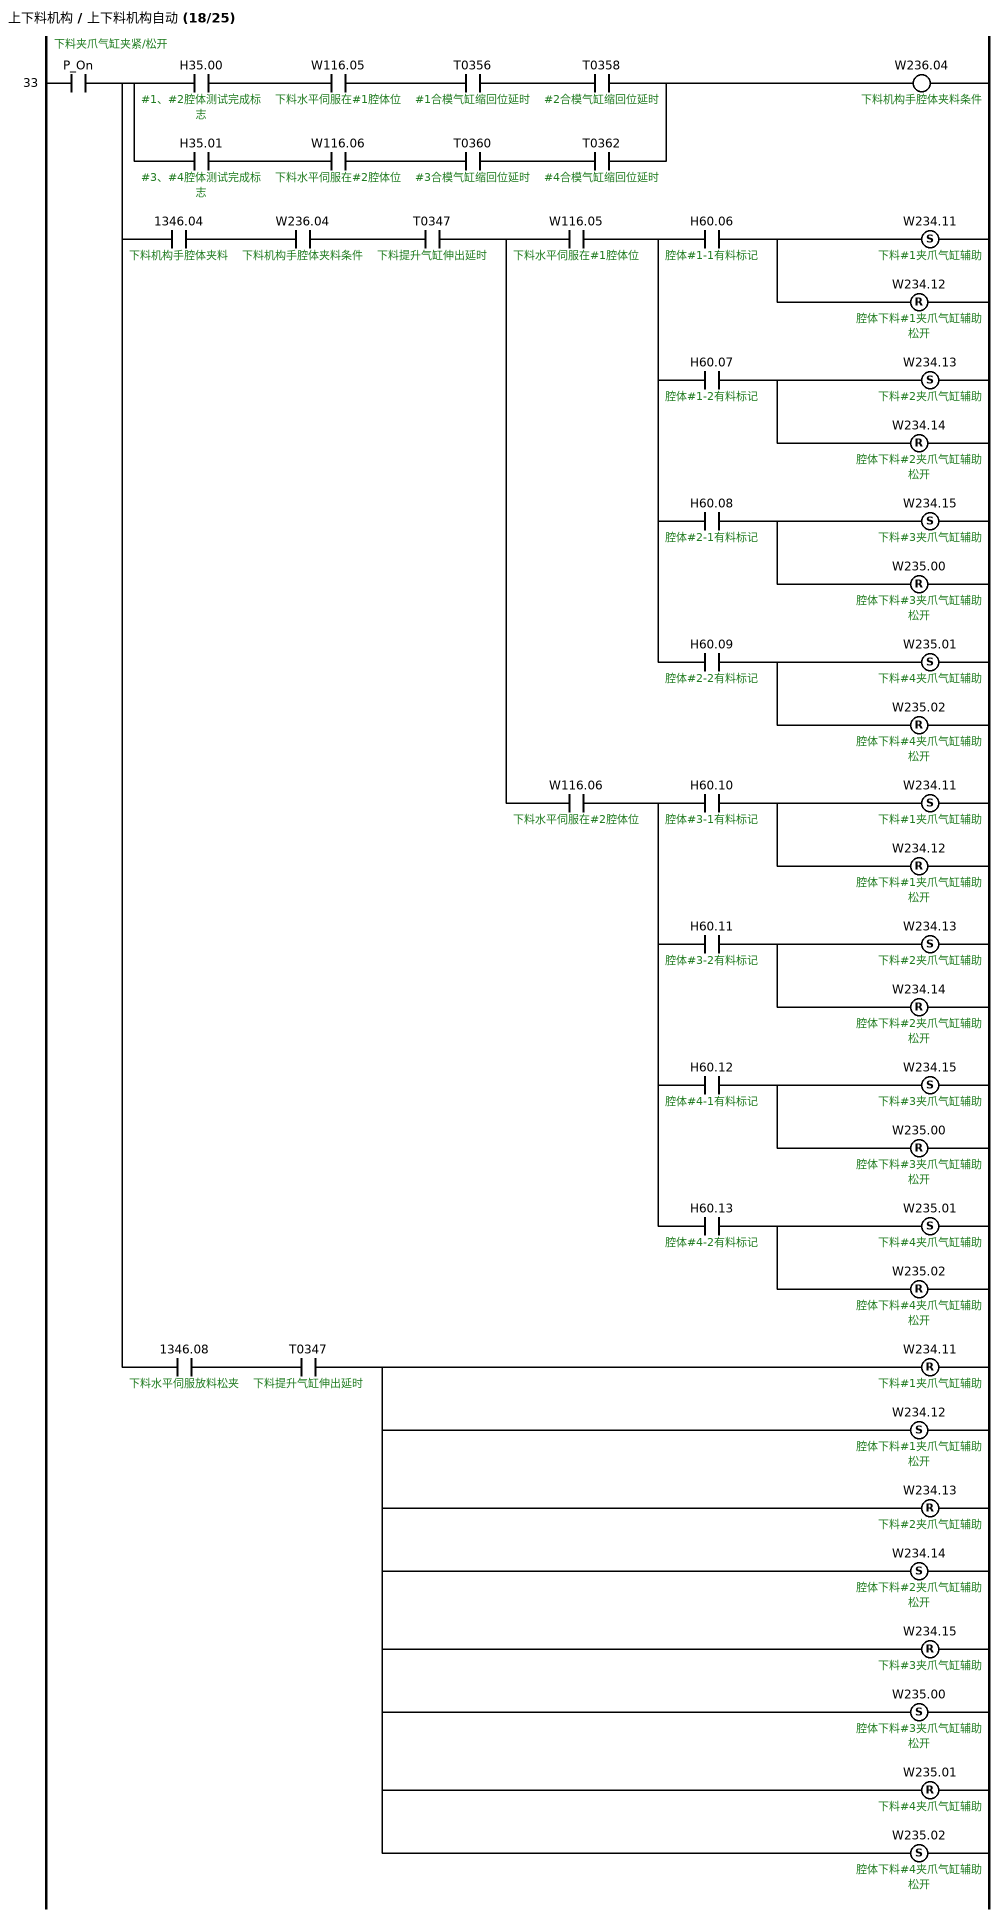
; rung 33: 下料夹爪气缸夹紧/松开
LD P_On
OUT TR0
LD H35.00  ; #1、#2腔体测试完成标志
AND W116.05  ; 下料水平伺服在#1腔体位
AND T0356  ; #1合模气缸缩回位延时
AND T0358  ; #2合模气缸缩回位延时
LD H35.01  ; #3、#4腔体测试完成标志
AND W116.06  ; 下料水平伺服在#2腔体位
AND T0360  ; #3合模气缸缩回位延时
AND T0362  ; #4合模气缸缩回位延时
ORLD
ANDLD
OUT W236.04  ; 下料机构手腔体夹料条件
LD TR0
AND 1346.04  ; 下料机构手腔体夹料
AND W236.04  ; 下料机构手腔体夹料条件
AND T0347  ; 下料提升气缸伸出延时
OUT TR1
AND W116.05  ; 下料水平伺服在#1腔体位
OUT TR2
AND H60.06  ; 腔体#1-1有料标记
SET W234.11  ; 下料#1夹爪气缸辅助
RSET W234.12  ; 腔体下料#1夹爪气缸辅助松开
LD TR2
AND H60.07  ; 腔体#1-2有料标记
SET W234.13  ; 下料#2夹爪气缸辅助
RSET W234.14  ; 腔体下料#2夹爪气缸辅助松开
LD TR2
AND H60.08  ; 腔体#2-1有料标记
SET W234.15  ; 下料#3夹爪气缸辅助
RSET W235.00  ; 腔体下料#3夹爪气缸辅助松开
LD TR2
AND H60.09  ; 腔体#2-2有料标记
SET W235.01  ; 下料#4夹爪气缸辅助
RSET W235.02  ; 腔体下料#4夹爪气缸辅助松开
LD TR1
AND W116.06  ; 下料水平伺服在#2腔体位
OUT TR1
AND H60.10  ; 腔体#3-1有料标记
SET W234.11  ; 下料#1夹爪气缸辅助
RSET W234.12  ; 腔体下料#1夹爪气缸辅助松开
LD TR1
AND H60.11  ; 腔体#3-2有料标记
SET W234.13  ; 下料#2夹爪气缸辅助
RSET W234.14  ; 腔体下料#2夹爪气缸辅助松开
LD TR1
AND H60.12  ; 腔体#4-1有料标记
SET W234.15  ; 下料#3夹爪气缸辅助
RSET W235.00  ; 腔体下料#3夹爪气缸辅助松开
LD TR1
AND H60.13  ; 腔体#4-2有料标记
SET W235.01  ; 下料#4夹爪气缸辅助
RSET W235.02  ; 腔体下料#4夹爪气缸辅助松开
LD TR0
AND 1346.08  ; 下料水平伺服放料松夹
AND T0347  ; 下料提升气缸伸出延时
RSET W234.11  ; 下料#1夹爪气缸辅助
SET W234.12  ; 腔体下料#1夹爪气缸辅助松开
RSET W234.13  ; 下料#2夹爪气缸辅助
SET W234.14  ; 腔体下料#2夹爪气缸辅助松开
RSET W234.15  ; 下料#3夹爪气缸辅助
SET W235.00  ; 腔体下料#3夹爪气缸辅助松开
RSET W235.01  ; 下料#4夹爪气缸辅助
SET W235.02  ; 腔体下料#4夹爪气缸辅助松开

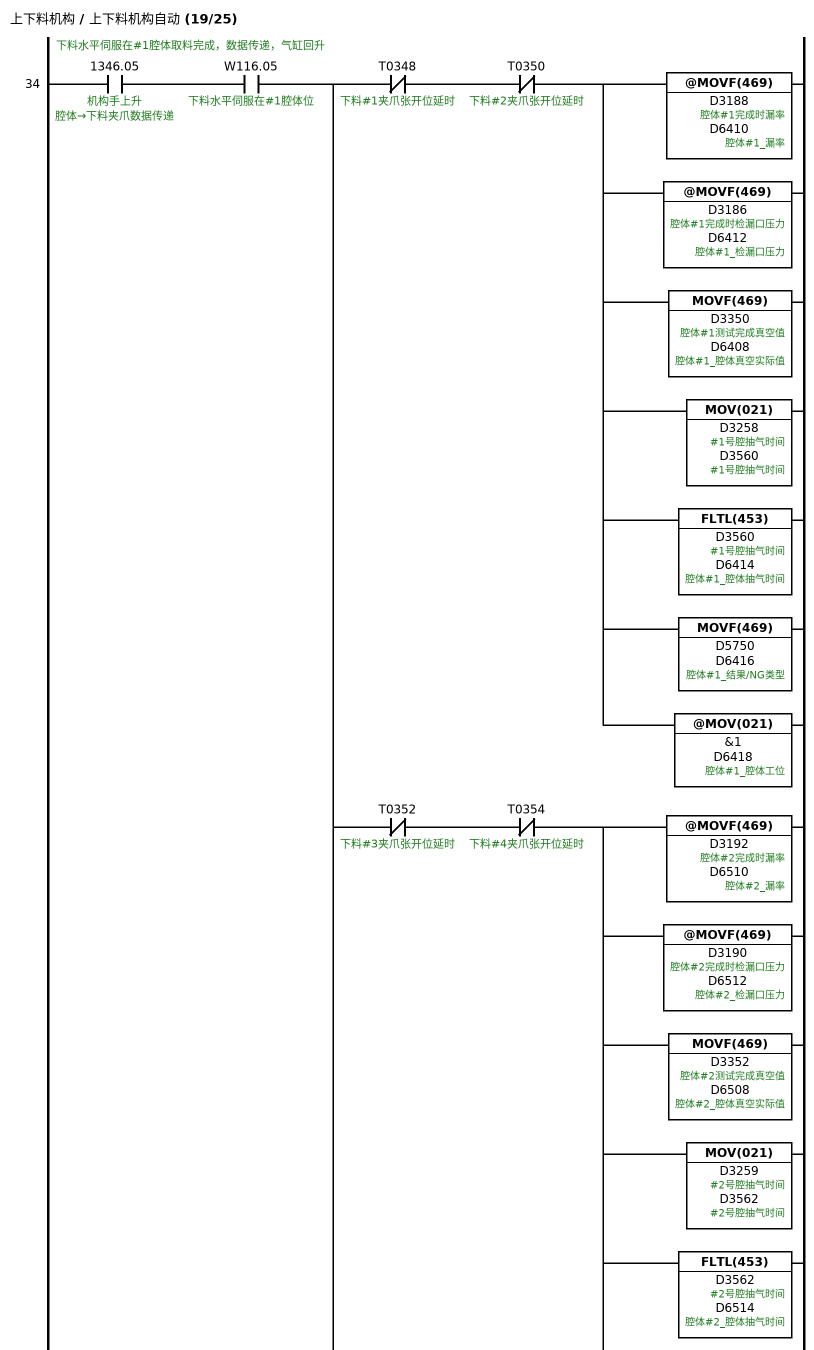

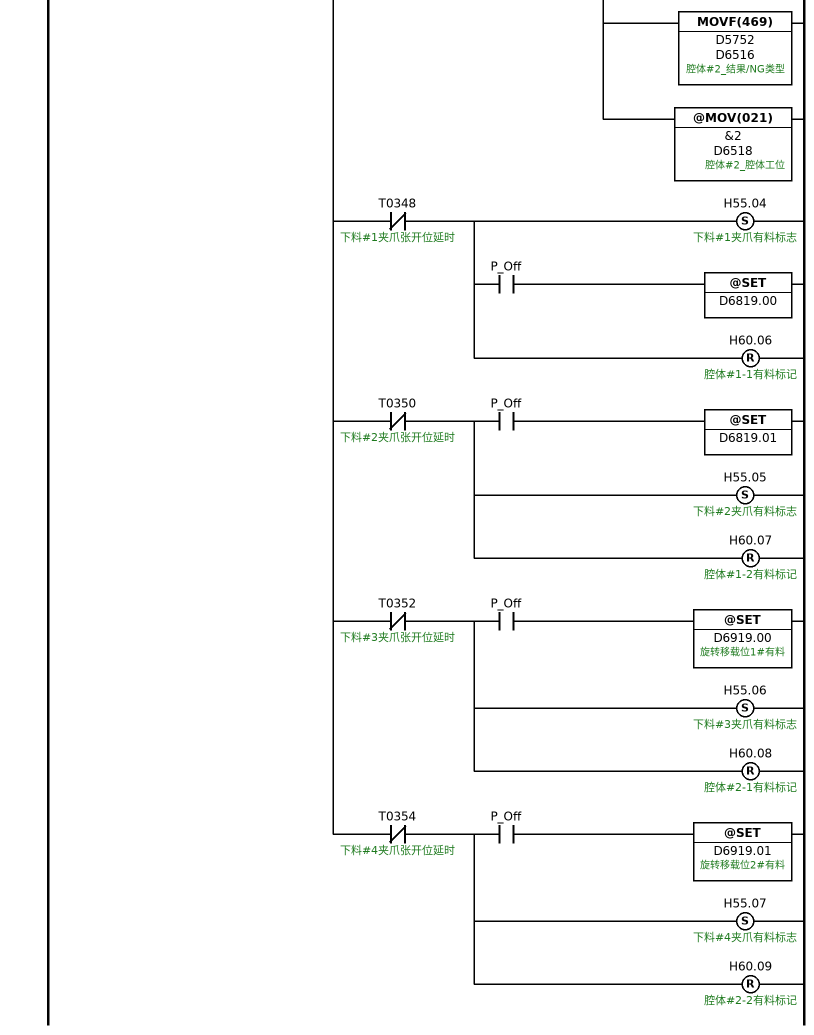
; rung 34: 下料水平伺服在#1腔体取料完成，数据传递，气缸回升
LD 1346.05  ; 机构手上升 腔体→下料夹爪数据传递
AND W116.05  ; 下料水平伺服在#1腔体位
OUT TR0
ANDNOT T0348  ; 下料#1夹爪张开位延时
ANDNOT T0350  ; 下料#2夹爪张开位延时
@MOVF(469) D3188 D6410  ; 腔体#1完成时漏率, 腔体#1_漏率
@MOVF(469) D3186 D6412  ; 腔体#1完成时检漏口压力, 腔体#1_检漏口压力
MOVF(469) D3350 D6408  ; 腔体#1测试完成真空值, 腔体#1_腔体真空实际值
MOV(021) D3258 D3560  ; #1号腔抽气时间
FLTL(453) D3560 D6414  ; #1号腔抽气时间, 腔体#1_腔体抽气时间
MOVF(469) D5750 D6416  ; 腔体#1_结果/NG类型
@MOV(021) &1 D6418  ; 腔体#1_腔体工位
LD TR0
ANDNOT T0352  ; 下料#3夹爪张开位延时
ANDNOT T0354  ; 下料#4夹爪张开位延时
@MOVF(469) D3192 D6510  ; 腔体#2完成时漏率, 腔体#2_漏率
@MOVF(469) D3190 D6512  ; 腔体#2完成时检漏口压力, 腔体#2_检漏口压力
MOVF(469) D3352 D6508  ; 腔体#2测试完成真空值, 腔体#2_腔体真空实际值
MOV(021) D3259 D3562  ; #2号腔抽气时间
FLTL(453) D3562 D6514  ; #2号腔抽气时间, 腔体#2_腔体抽气时间
MOVF(469) D5752 D6516  ; 腔体#2_结果/NG类型
@MOV(021) &2 D6518  ; 腔体#2_腔体工位
LD TR0
ANDNOT T0348  ; 下料#1夹爪张开位延时
OUT TR1
SET H55.04  ; 下料#1夹爪有料标志
AND P_Off
@SET D6819.00
LD TR1
RSET H60.06  ; 腔体#1-1有料标记
LD TR0
ANDNOT T0350  ; 下料#2夹爪张开位延时
OUT TR1
AND P_Off
@SET D6819.01
LD TR1
SET H55.05  ; 下料#2夹爪有料标志
RSET H60.07  ; 腔体#1-2有料标记
LD TR0
ANDNOT T0352  ; 下料#3夹爪张开位延时
OUT TR1
AND P_Off
@SET D6919.00  ; 旋转移载位1#有料
LD TR1
SET H55.06  ; 下料#3夹爪有料标志
RSET H60.08  ; 腔体#2-1有料标记
LD TR0
ANDNOT T0354  ; 下料#4夹爪张开位延时
OUT TR0
AND P_Off
@SET D6919.01  ; 旋转移载位2#有料
LD TR0
SET H55.07  ; 下料#4夹爪有料标志
RSET H60.09  ; 腔体#2-2有料标记

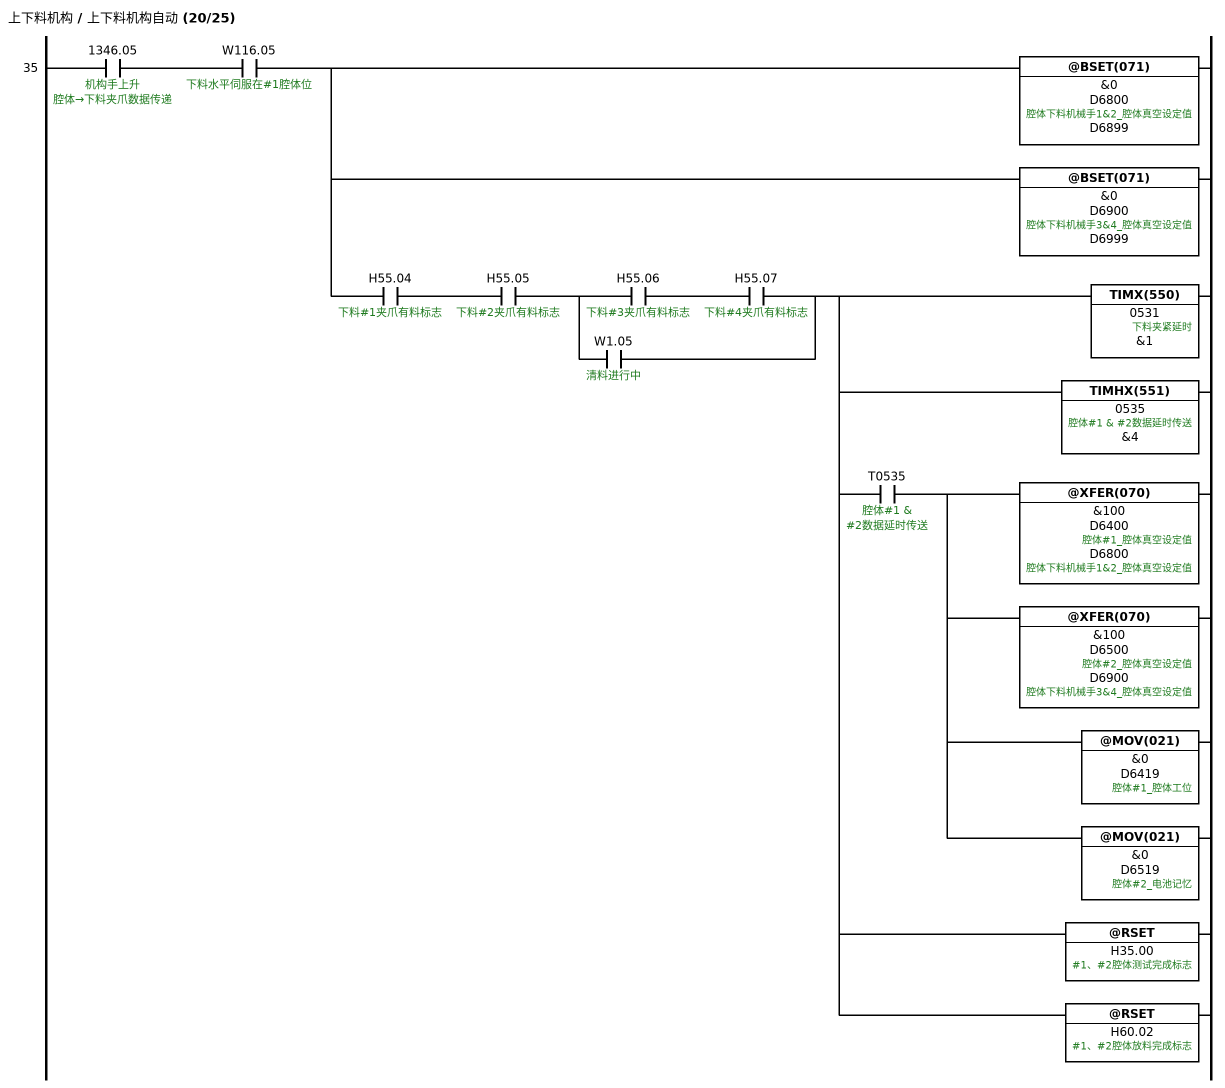
; rung 35
LD 1346.05  ; 机构手上升 腔体→下料夹爪数据传递
AND W116.05  ; 下料水平伺服在#1腔体位
@BSET(071) &0 D6800 D6899  ; 腔体下料机械手1&2_腔体真空设定值
@BSET(071) &0 D6900 D6999  ; 腔体下料机械手3&4_腔体真空设定值
AND H55.04  ; 下料#1夹爪有料标志
AND H55.05  ; 下料#2夹爪有料标志
LD H55.06  ; 下料#3夹爪有料标志
AND H55.07  ; 下料#4夹爪有料标志
OR W1.05  ; 清料进行中
ANDLD
OUT TR0
TIMX(550) 0531 &1  ; 下料夹紧延时
TIMHX(551) 0535 &4  ; 腔体#1 & #2数据延时传送
AND T0535  ; 腔体#1 & #2数据延时传送
@XFER(070) &100 D6400 D6800  ; 腔体#1_腔体真空设定值, 腔体下料机械手1&2_腔体真空设定值
@XFER(070) &100 D6500 D6900  ; 腔体#2_腔体真空设定值, 腔体下料机械手3&4_腔体真空设定值
@MOV(021) &0 D6419  ; 腔体#1_腔体工位
@MOV(021) &0 D6519  ; 腔体#2_电池记忆
LD TR0
@RSET H35.00  ; #1、#2腔体测试完成标志
@RSET H60.02  ; #1、#2腔体放料完成标志

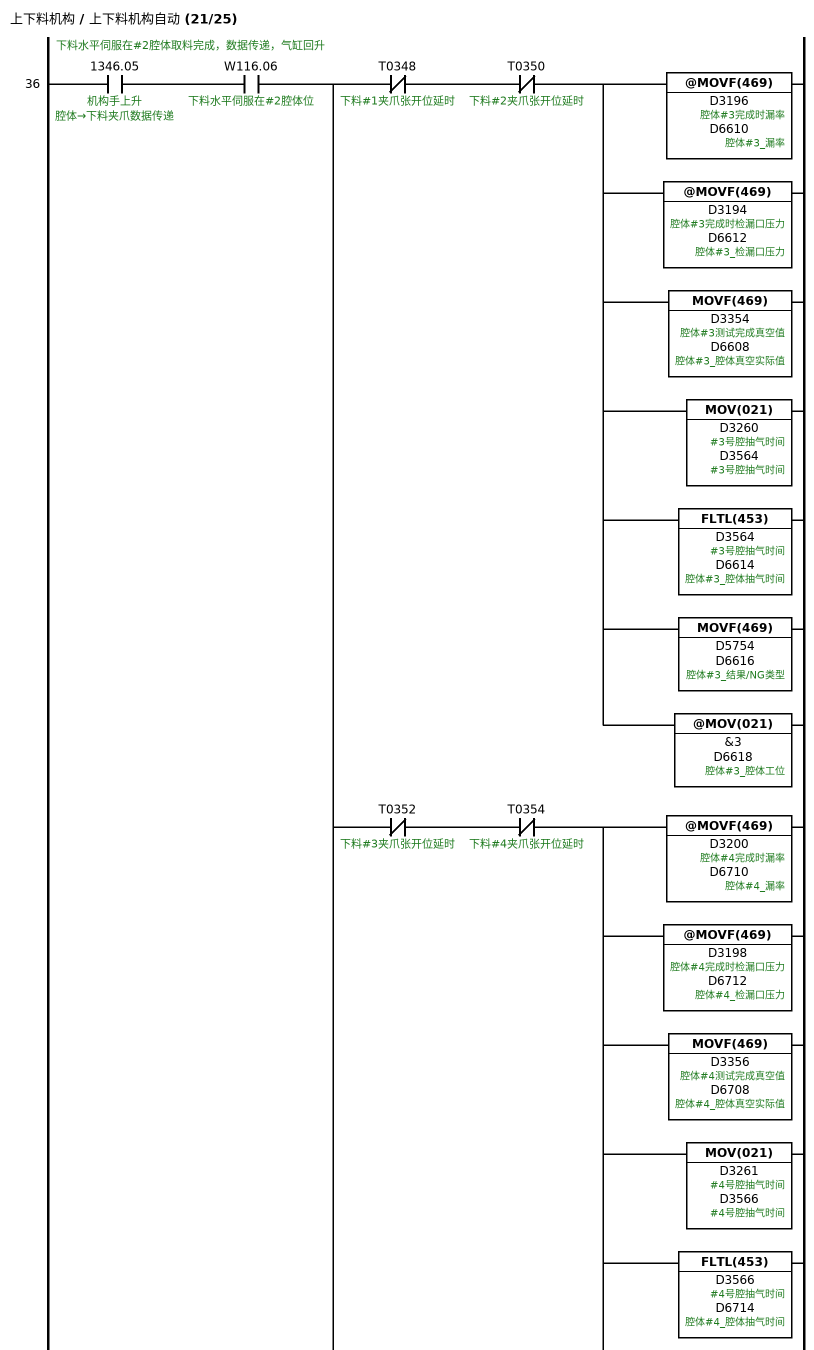

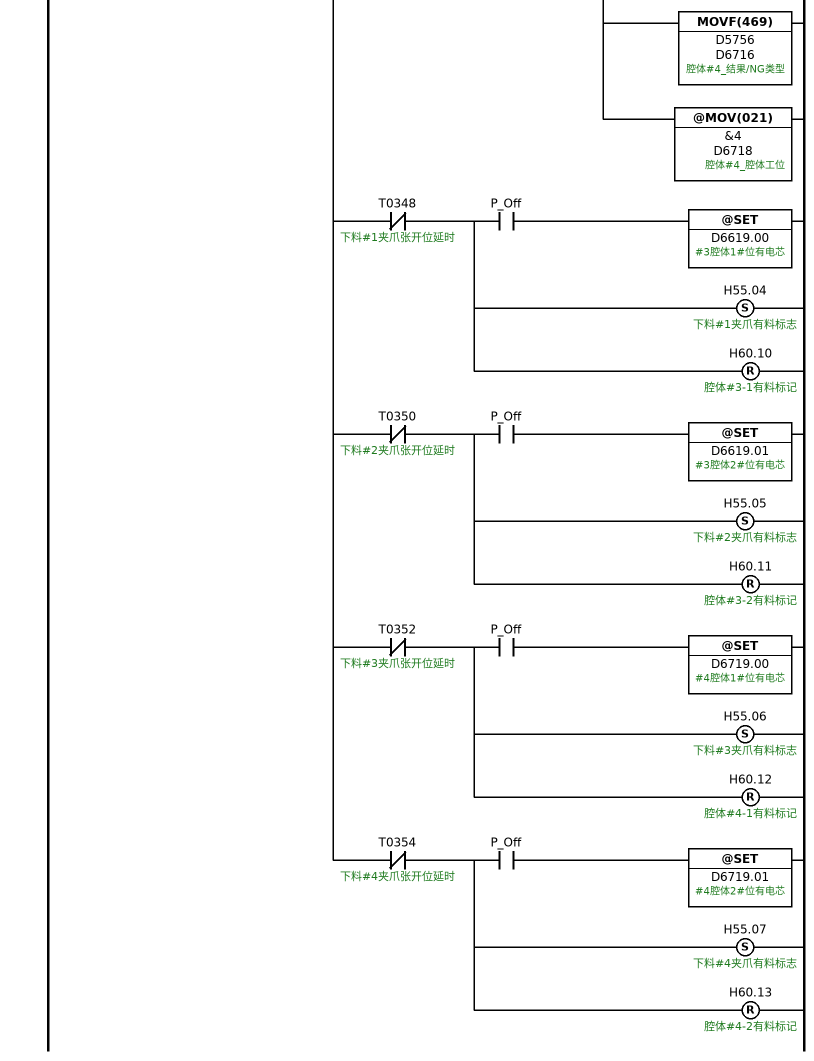
; rung 36: 下料水平伺服在#2腔体取料完成，数据传递，气缸回升
LD 1346.05  ; 机构手上升 腔体→下料夹爪数据传递
AND W116.06  ; 下料水平伺服在#2腔体位
OUT TR0
ANDNOT T0348  ; 下料#1夹爪张开位延时
ANDNOT T0350  ; 下料#2夹爪张开位延时
@MOVF(469) D3196 D6610  ; 腔体#3完成时漏率, 腔体#3_漏率
@MOVF(469) D3194 D6612  ; 腔体#3完成时检漏口压力, 腔体#3_检漏口压力
MOVF(469) D3354 D6608  ; 腔体#3测试完成真空值, 腔体#3_腔体真空实际值
MOV(021) D3260 D3564  ; #3号腔抽气时间
FLTL(453) D3564 D6614  ; #3号腔抽气时间, 腔体#3_腔体抽气时间
MOVF(469) D5754 D6616  ; 腔体#3_结果/NG类型
@MOV(021) &3 D6618  ; 腔体#3_腔体工位
LD TR0
ANDNOT T0352  ; 下料#3夹爪张开位延时
ANDNOT T0354  ; 下料#4夹爪张开位延时
@MOVF(469) D3200 D6710  ; 腔体#4完成时漏率, 腔体#4_漏率
@MOVF(469) D3198 D6712  ; 腔体#4完成时检漏口压力, 腔体#4_检漏口压力
MOVF(469) D3356 D6708  ; 腔体#4测试完成真空值, 腔体#4_腔体真空实际值
MOV(021) D3261 D3566  ; #4号腔抽气时间
FLTL(453) D3566 D6714  ; #4号腔抽气时间, 腔体#4_腔体抽气时间
MOVF(469) D5756 D6716  ; 腔体#4_结果/NG类型
@MOV(021) &4 D6718  ; 腔体#4_腔体工位
LD TR0
ANDNOT T0348  ; 下料#1夹爪张开位延时
OUT TR1
AND P_Off
@SET D6619.00  ; #3腔体1#位有电芯
LD TR1
SET H55.04  ; 下料#1夹爪有料标志
RSET H60.10  ; 腔体#3-1有料标记
LD TR0
ANDNOT T0350  ; 下料#2夹爪张开位延时
OUT TR1
AND P_Off
@SET D6619.01  ; #3腔体2#位有电芯
LD TR1
SET H55.05  ; 下料#2夹爪有料标志
RSET H60.11  ; 腔体#3-2有料标记
LD TR0
ANDNOT T0352  ; 下料#3夹爪张开位延时
OUT TR1
AND P_Off
@SET D6719.00  ; #4腔体1#位有电芯
LD TR1
SET H55.06  ; 下料#3夹爪有料标志
RSET H60.12  ; 腔体#4-1有料标记
LD TR0
ANDNOT T0354  ; 下料#4夹爪张开位延时
OUT TR0
AND P_Off
@SET D6719.01  ; #4腔体2#位有电芯
LD TR0
SET H55.07  ; 下料#4夹爪有料标志
RSET H60.13  ; 腔体#4-2有料标记

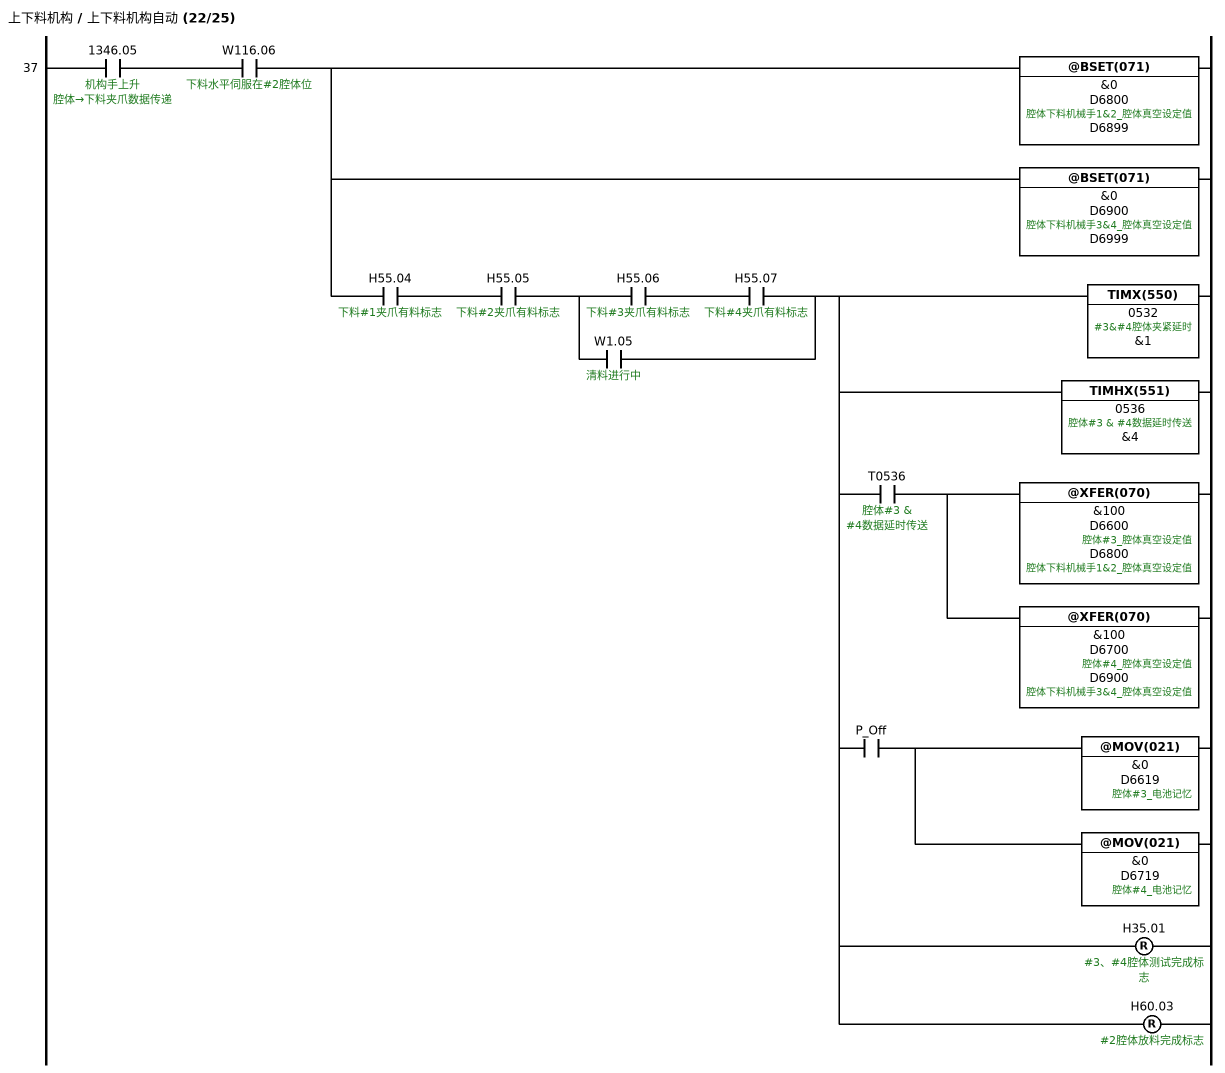
; rung 37
LD 1346.05  ; 机构手上升 腔体→下料夹爪数据传递
AND W116.06  ; 下料水平伺服在#2腔体位
@BSET(071) &0 D6800 D6899  ; 腔体下料机械手1&2_腔体真空设定值
@BSET(071) &0 D6900 D6999  ; 腔体下料机械手3&4_腔体真空设定值
AND H55.04  ; 下料#1夹爪有料标志
AND H55.05  ; 下料#2夹爪有料标志
LD H55.06  ; 下料#3夹爪有料标志
AND H55.07  ; 下料#4夹爪有料标志
OR W1.05  ; 清料进行中
ANDLD
OUT TR0
TIMX(550) 0532 &1  ; #3&#4腔体夹紧延时
TIMHX(551) 0536 &4  ; 腔体#3 & #4数据延时传送
AND T0536  ; 腔体#3 & #4数据延时传送
@XFER(070) &100 D6600 D6800  ; 腔体#3_腔体真空设定值, 腔体下料机械手1&2_腔体真空设定值
@XFER(070) &100 D6700 D6900  ; 腔体#4_腔体真空设定值, 腔体下料机械手3&4_腔体真空设定值
LD TR0
AND P_Off
@MOV(021) &0 D6619  ; 腔体#3_电池记忆
@MOV(021) &0 D6719  ; 腔体#4_电池记忆
LD TR0
RSET H35.01  ; #3、#4腔体测试完成标志
RSET H60.03  ; #2腔体放料完成标志

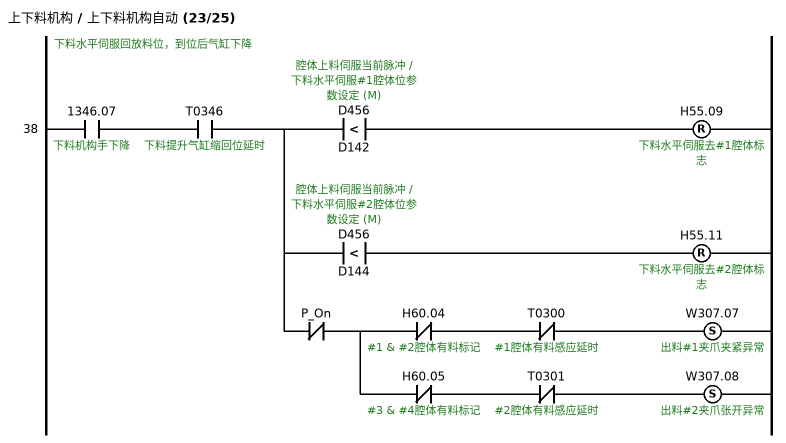
; rung 38: 下料水平伺服回放料位，到位后气缸下降
LD 1346.07  ; 下料机构手下降
AND T0346  ; 下料提升气缸缩回位延时
OUT TR0
AND<F(331) D456 D142  ; 腔体上料伺服当前脉冲, 下料水平伺服#1腔体位参数设定 (M)
RSET H55.09  ; 下料水平伺服去#1腔体标志
LD TR0
AND<F(331) D456 D144  ; 腔体上料伺服当前脉冲, 下料水平伺服#2腔体位参数设定 (M)
RSET H55.11  ; 下料水平伺服去#2腔体标志
LD TR0
ANDNOT P_On
OUT TR0
ANDNOT H60.04  ; #1 & #2腔体有料标记
ANDNOT T0300  ; #1腔体有料感应延时
SET W307.07  ; 出料#1夹爪夹紧异常
LD TR0
ANDNOT H60.05  ; #3 & #4腔体有料标记
ANDNOT T0301  ; #2腔体有料感应延时
SET W307.08  ; 出料#2夹爪张开异常

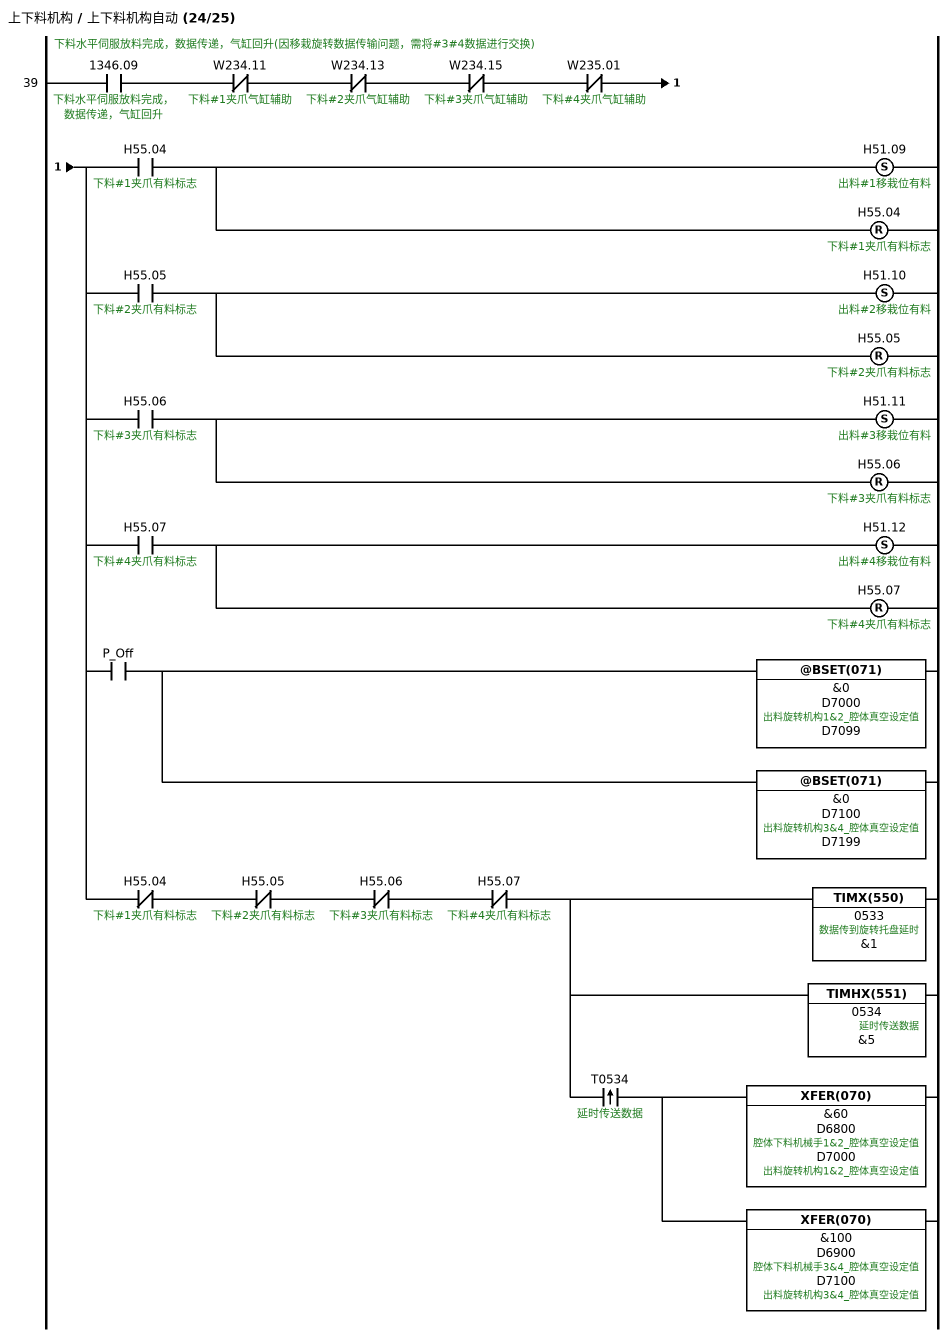
; rung 39: 下料水平伺服放料完成，数据传递，气缸回升(因移栽旋转数据传输问题，需将#3#4数据进行交换)
LD 1346.09  ; 下料水平伺服放料完成，数据传递，气缸回升
ANDNOT W234.11  ; 下料#1夹爪气缸辅助
ANDNOT W234.13  ; 下料#2夹爪气缸辅助
ANDNOT W234.15  ; 下料#3夹爪气缸辅助
ANDNOT W235.01  ; 下料#4夹爪气缸辅助
OUT TR0
AND H55.04  ; 下料#1夹爪有料标志
SET H51.09  ; 出料#1移栽位有料
RSET H55.04  ; 下料#1夹爪有料标志
LD TR0
AND H55.05  ; 下料#2夹爪有料标志
SET H51.10  ; 出料#2移栽位有料
RSET H55.05  ; 下料#2夹爪有料标志
LD TR0
AND H55.06  ; 下料#3夹爪有料标志
SET H51.11  ; 出料#3移栽位有料
RSET H55.06  ; 下料#3夹爪有料标志
LD TR0
AND H55.07  ; 下料#4夹爪有料标志
SET H51.12  ; 出料#4移栽位有料
RSET H55.07  ; 下料#4夹爪有料标志
LD TR0
AND P_Off
@BSET(071) &0 D7000 D7099  ; 出料旋转机构1&2_腔体真空设定值
@BSET(071) &0 D7100 D7199  ; 出料旋转机构3&4_腔体真空设定值
LD TR0
ANDNOT H55.04  ; 下料#1夹爪有料标志
ANDNOT H55.05  ; 下料#2夹爪有料标志
ANDNOT H55.06  ; 下料#3夹爪有料标志
ANDNOT H55.07  ; 下料#4夹爪有料标志
TIMX(550) 0533 &1  ; 数据传到旋转托盘延时
TIMHX(551) 0534 &5  ; 延时传送数据
@AND T0534  ; 延时传送数据
XFER(070) &60 D6800 D7000  ; 腔体下料机械手1&2_腔体真空设定值, 出料旋转机构1&2_腔体真空设定值
XFER(070) &100 D6900 D7100  ; 腔体下料机械手3&4_腔体真空设定值, 出料旋转机构3&4_腔体真空设定值

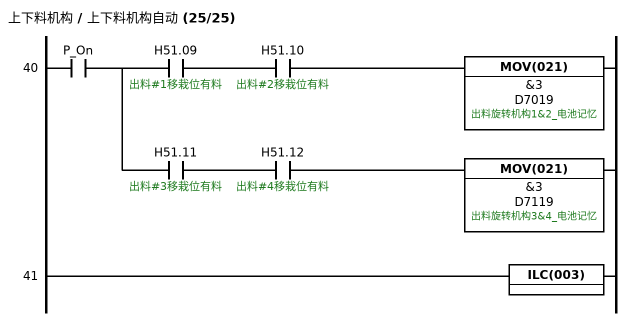
; rung 40
LD P_On
OUT TR0
AND H51.09  ; 出料#1移栽位有料
AND H51.10  ; 出料#2移栽位有料
MOV(021) &3 D7019  ; 出料旋转机构1&2_电池记忆
LD TR0
AND H51.11  ; 出料#3移栽位有料
AND H51.12  ; 出料#4移栽位有料
MOV(021) &3 D7119  ; 出料旋转机构3&4_电池记忆
; rung 41
ILC(003)

### Section 上下料机构手动

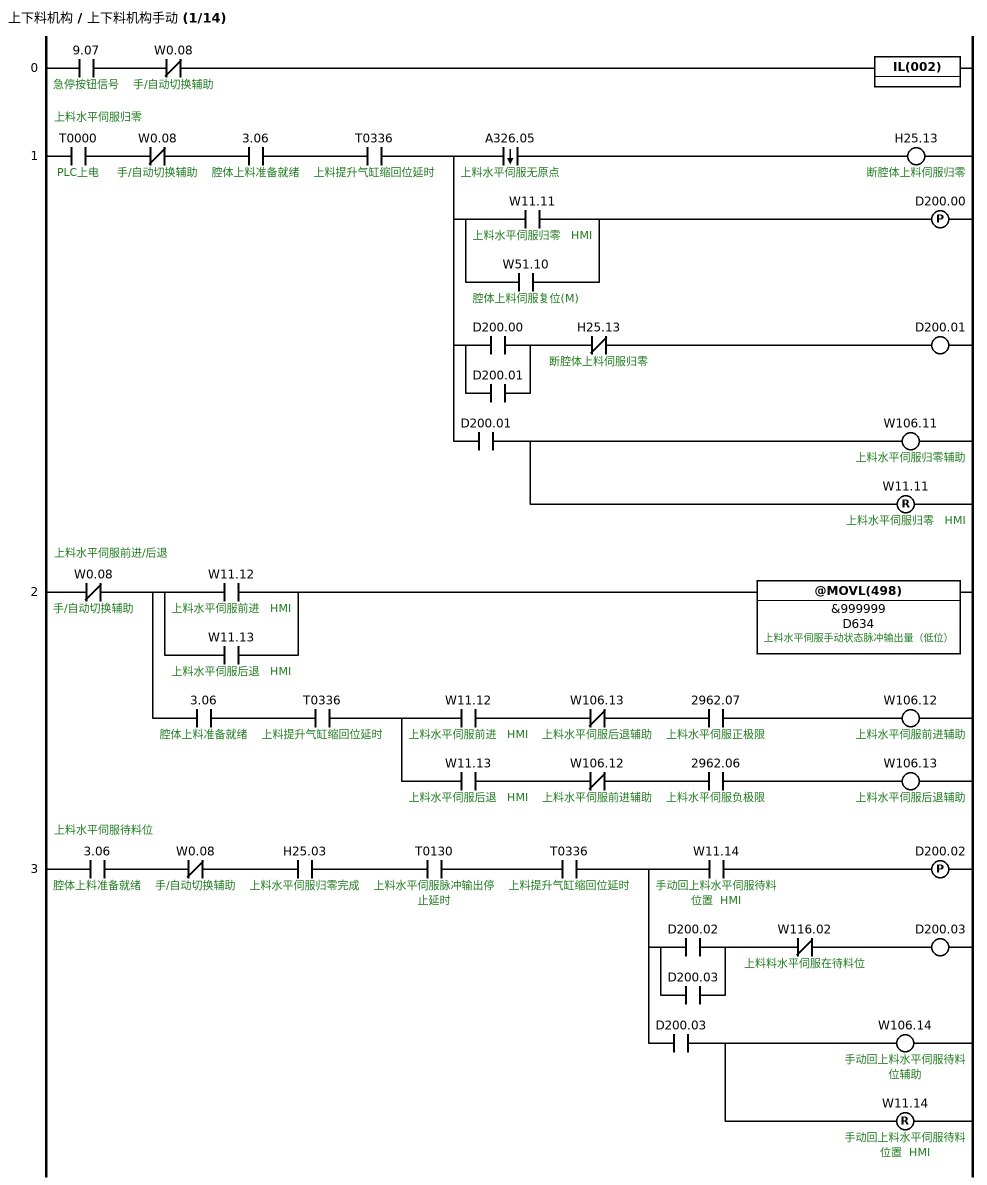
; rung 0
LD 9.07  ; 急停按钮信号
ANDNOT W0.08  ; 手/自动切换辅助
IL(002)
; rung 1: 上料水平伺服归零
LD T0000  ; PLC上电
ANDNOT W0.08  ; 手/自动切换辅助
AND 3.06  ; 腔体上料准备就绪
AND T0336  ; 上料提升气缸缩回位延时
OUT TR0
%AND A326.05  ; 上料水平伺服无原点
OUT H25.13  ; 断腔体上料伺服归零
LD TR0
LD W11.11  ; 上料水平伺服归零   HMI
OR W51.10  ; 腔体上料伺服复位(M)
ANDLD
DIFU(013) D200.00
LD TR0
LD D200.00
OR D200.01
ANDLD
ANDNOT H25.13  ; 断腔体上料伺服归零
OUT D200.01
LD TR0
AND D200.01
OUT W106.11  ; 上料水平伺服归零辅助
RSET W11.11  ; 上料水平伺服归零   HMI
; rung 2: 上料水平伺服前进/后退
LDNOT W0.08  ; 手/自动切换辅助
OUT TR0
LD W11.12  ; 上料水平伺服前进   HMI
OR W11.13  ; 上料水平伺服后退   HMI
ANDLD
@MOVL(498) &999999 D634  ; 上料水平伺服手动状态脉冲输出量（低位）
LD TR0
AND 3.06  ; 腔体上料准备就绪
AND T0336  ; 上料提升气缸缩回位延时
OUT TR0
AND W11.12  ; 上料水平伺服前进   HMI
ANDNOT W106.13  ; 上料水平伺服后退辅助
AND 2962.07  ; 上料水平伺服正极限
OUT W106.12  ; 上料水平伺服前进辅助
LD TR0
AND W11.13  ; 上料水平伺服后退   HMI
ANDNOT W106.12  ; 上料水平伺服前进辅助
AND 2962.06  ; 上料水平伺服负极限
OUT W106.13  ; 上料水平伺服后退辅助
; rung 3: 上料水平伺服待料位
LD 3.06  ; 腔体上料准备就绪
ANDNOT W0.08  ; 手/自动切换辅助
AND H25.03  ; 上料水平伺服归零完成
AND T0130  ; 上料水平伺服脉冲输出停止延时
AND T0336  ; 上料提升气缸缩回位延时
OUT TR0
AND W11.14  ; 手动回上料水平伺服待料位置  HMI
DIFU(013) D200.02
LD TR0
LD D200.02
OR D200.03
ANDLD
ANDNOT W116.02  ; 上料料水平伺服在待料位
OUT D200.03
LD TR0
AND D200.03
OUT W106.14  ; 手动回上料水平伺服待料位辅助
RSET W11.14  ; 手动回上料水平伺服待料位置  HMI

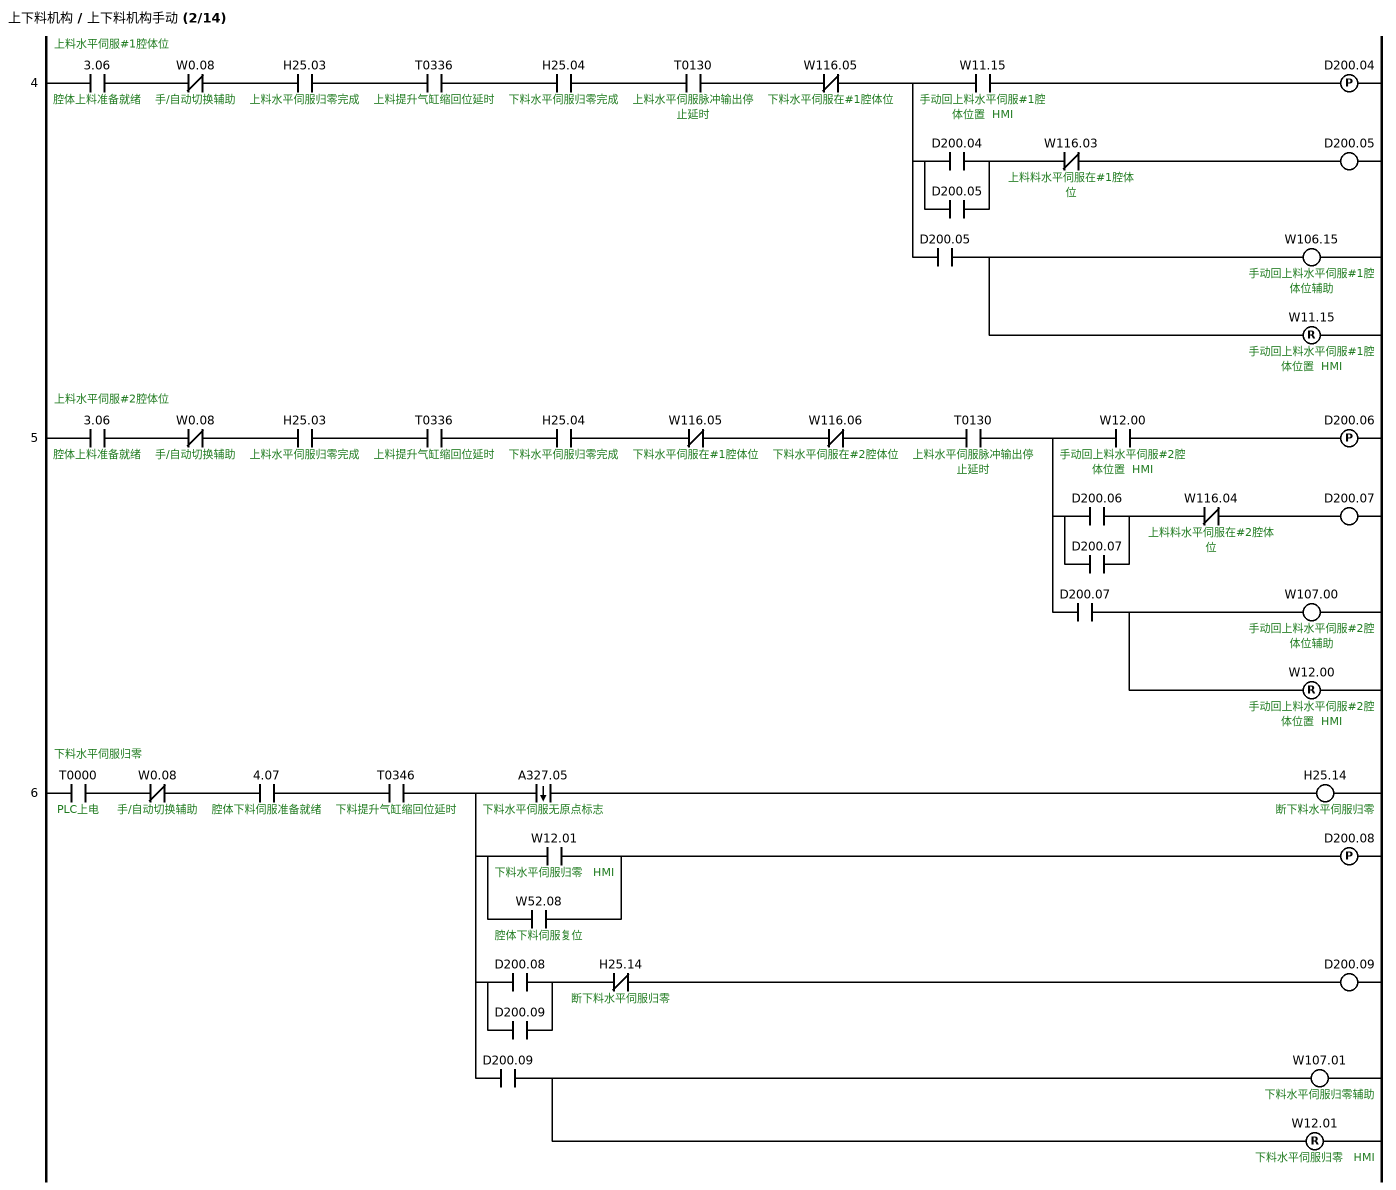
; rung 4: 上料水平伺服#1腔体位
LD 3.06  ; 腔体上料准备就绪
ANDNOT W0.08  ; 手/自动切换辅助
AND H25.03  ; 上料水平伺服归零完成
AND T0336  ; 上料提升气缸缩回位延时
AND H25.04  ; 下料水平伺服归零完成
AND T0130  ; 上料水平伺服脉冲输出停止延时
ANDNOT W116.05  ; 下料水平伺服在#1腔体位
OUT TR0
AND W11.15  ; 手动回上料水平伺服#1腔体位置  HMI
DIFU(013) D200.04
LD TR0
LD D200.04
OR D200.05
ANDLD
ANDNOT W116.03  ; 上料料水平伺服在#1腔体位
OUT D200.05
LD TR0
AND D200.05
OUT W106.15  ; 手动回上料水平伺服#1腔体位辅助
RSET W11.15  ; 手动回上料水平伺服#1腔体位置  HMI
; rung 5: 上料水平伺服#2腔体位
LD 3.06  ; 腔体上料准备就绪
ANDNOT W0.08  ; 手/自动切换辅助
AND H25.03  ; 上料水平伺服归零完成
AND T0336  ; 上料提升气缸缩回位延时
AND H25.04  ; 下料水平伺服归零完成
ANDNOT W116.05  ; 下料水平伺服在#1腔体位
ANDNOT W116.06  ; 下料水平伺服在#2腔体位
AND T0130  ; 上料水平伺服脉冲输出停止延时
OUT TR0
AND W12.00  ; 手动回上料水平伺服#2腔体位置  HMI
DIFU(013) D200.06
LD TR0
LD D200.06
OR D200.07
ANDLD
ANDNOT W116.04  ; 上料料水平伺服在#2腔体位
OUT D200.07
LD TR0
AND D200.07
OUT W107.00  ; 手动回上料水平伺服#2腔体位辅助
RSET W12.00  ; 手动回上料水平伺服#2腔体位置  HMI
; rung 6: 下料水平伺服归零
LD T0000  ; PLC上电
ANDNOT W0.08  ; 手/自动切换辅助
AND 4.07  ; 腔体下料伺服准备就绪
AND T0346  ; 下料提升气缸缩回位延时
OUT TR0
%AND A327.05  ; 下料水平伺服无原点标志
OUT H25.14  ; 断下料水平伺服归零
LD TR0
LD W12.01  ; 下料水平伺服归零   HMI
OR W52.08  ; 腔体下料伺服复位
ANDLD
DIFU(013) D200.08
LD TR0
LD D200.08
OR D200.09
ANDLD
ANDNOT H25.14  ; 断下料水平伺服归零
OUT D200.09
LD TR0
AND D200.09
OUT W107.01  ; 下料水平伺服归零辅助
RSET W12.01  ; 下料水平伺服归零   HMI

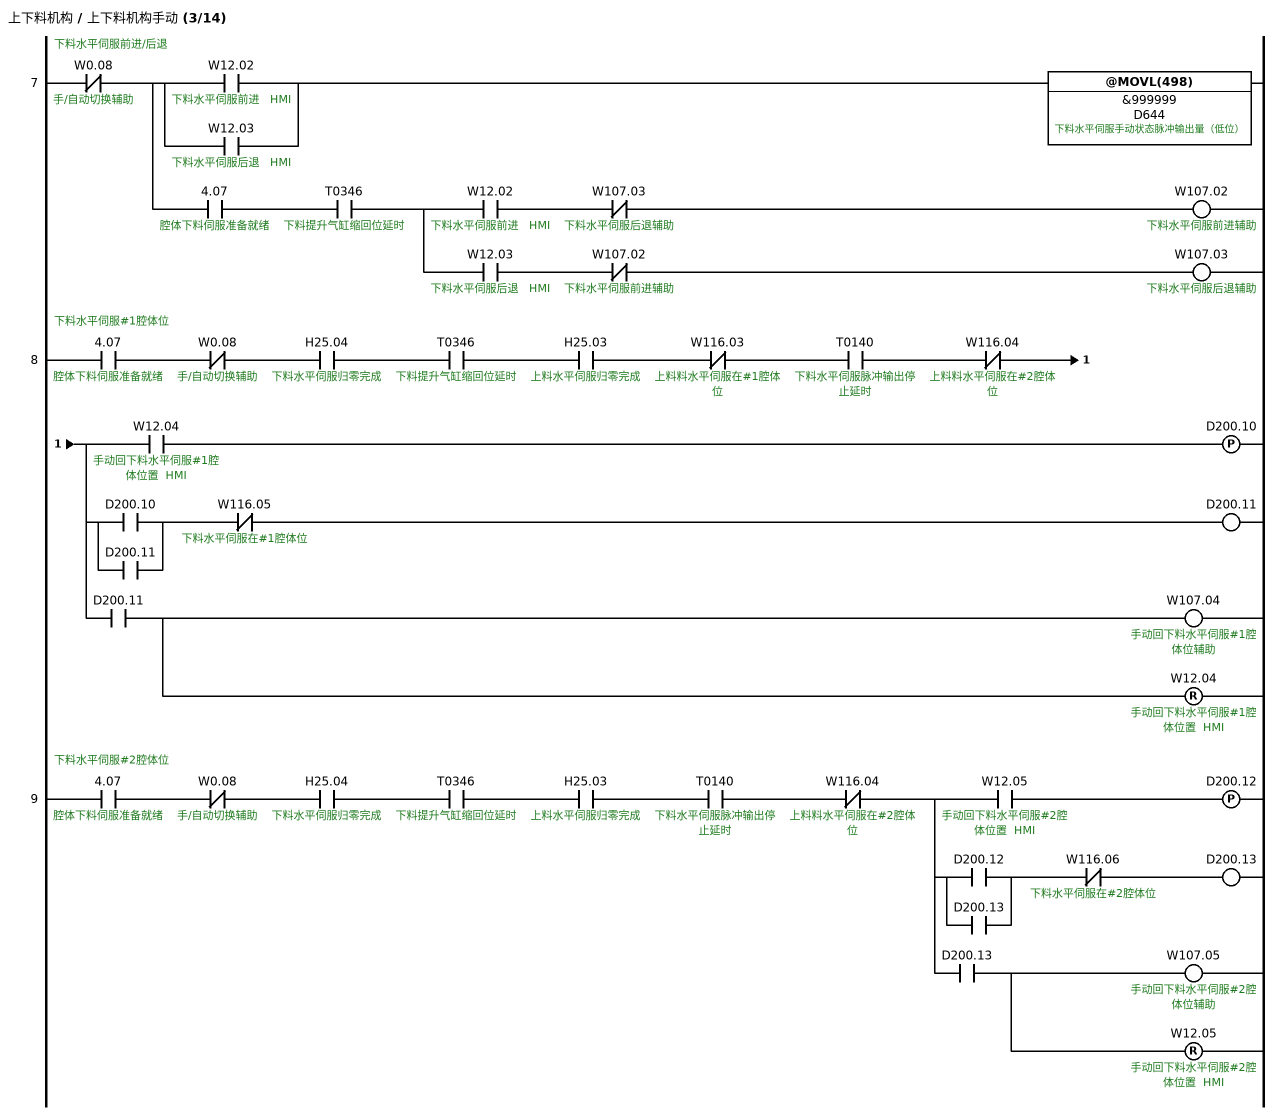
; rung 7: 下料水平伺服前进/后退
LDNOT W0.08  ; 手/自动切换辅助
OUT TR0
LD W12.02  ; 下料水平伺服前进   HMI
OR W12.03  ; 下料水平伺服后退   HMI
ANDLD
@MOVL(498) &999999 D644  ; 下料水平伺服手动状态脉冲输出量（低位）
LD TR0
AND 4.07  ; 腔体下料伺服准备就绪
AND T0346  ; 下料提升气缸缩回位延时
OUT TR0
AND W12.02  ; 下料水平伺服前进   HMI
ANDNOT W107.03  ; 下料水平伺服后退辅助
OUT W107.02  ; 下料水平伺服前进辅助
LD TR0
AND W12.03  ; 下料水平伺服后退   HMI
ANDNOT W107.02  ; 下料水平伺服前进辅助
OUT W107.03  ; 下料水平伺服后退辅助
; rung 8: 下料水平伺服#1腔体位
LD 4.07  ; 腔体下料伺服准备就绪
ANDNOT W0.08  ; 手/自动切换辅助
AND H25.04  ; 下料水平伺服归零完成
AND T0346  ; 下料提升气缸缩回位延时
AND H25.03  ; 上料水平伺服归零完成
ANDNOT W116.03  ; 上料料水平伺服在#1腔体位
AND T0140  ; 下料水平伺服脉冲输出停止延时
ANDNOT W116.04  ; 上料料水平伺服在#2腔体位
OUT TR0
AND W12.04  ; 手动回下料水平伺服#1腔体位置  HMI
DIFU(013) D200.10
LD TR0
LD D200.10
OR D200.11
ANDLD
ANDNOT W116.05  ; 下料水平伺服在#1腔体位
OUT D200.11
LD TR0
AND D200.11
OUT W107.04  ; 手动回下料水平伺服#1腔体位辅助
RSET W12.04  ; 手动回下料水平伺服#1腔体位置  HMI
; rung 9: 下料水平伺服#2腔体位
LD 4.07  ; 腔体下料伺服准备就绪
ANDNOT W0.08  ; 手/自动切换辅助
AND H25.04  ; 下料水平伺服归零完成
AND T0346  ; 下料提升气缸缩回位延时
AND H25.03  ; 上料水平伺服归零完成
AND T0140  ; 下料水平伺服脉冲输出停止延时
ANDNOT W116.04  ; 上料料水平伺服在#2腔体位
OUT TR0
AND W12.05  ; 手动回下料水平伺服#2腔体位置  HMI
DIFU(013) D200.12
LD TR0
LD D200.12
OR D200.13
ANDLD
ANDNOT W116.06  ; 下料水平伺服在#2腔体位
OUT D200.13
LD TR0
AND D200.13
OUT W107.05  ; 手动回下料水平伺服#2腔体位辅助
RSET W12.05  ; 手动回下料水平伺服#2腔体位置  HMI

